ABB RAPID module: bbff74c6.mod

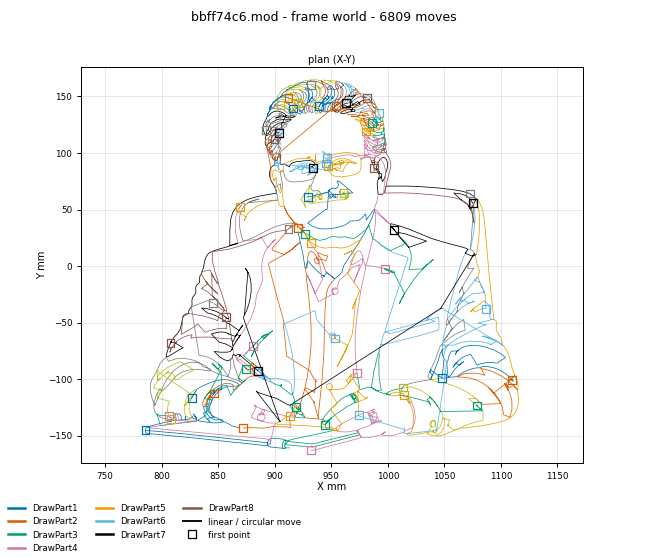
[picture p0: tool path of bbff74c6.mod in frame world, 6809 of 6811 moves have a stored position in this frame; points joined in program order, loops and branches not executed]
MODULE ImageDraw
  ! Generated 2026-10-07 06:23 for ABB IRB 1600-10/1.45: 764 strokes
  ! Page 500 x 350 mm. Work object wPaper: Z points up, so pen-up is +Z and the tool uses orientation [0,1,0,0].
  PERS tooldata tPen:=[TRUE,[[0,0,120],[1,0,0,0]],[0.3,[0,0,60],[1,0,0,0],0,0,0]];
  PERS wobjdata wPaper:=[FALSE,TRUE,"",[[700,-175,0],[1,0,0,0]],[[0,0,0],[1,0,0,0]]];
  CONST robtarget pOrigin:=[[0,0,0],[0,1,0,0],[0,0,0,0],[9E9,9E9,9E9,9E9,9E9,9E9]];
  CONST jointtarget jHome:=[[0,0,0,0,30,0],[9E9,9E9,9E9,9E9,9E9,9E9]];
  CONST speeddata vTravel:=[250,200,5000,1000];

  PROC DrawImage()
    SingArea\Wrist;
    ConfL\Off;
    ConfJ\Off;
    MoveAbsJ jHome\NoEOffs,vTravel,fine,tPen;
    DrawPart1;
    DrawPart2;
    DrawPart3;
    DrawPart4;
    DrawPart5;
    DrawPart6;
    DrawPart7;
    DrawPart8;
    DrawPart9;
    DrawPart10;
    DrawPart11;
    DrawPart12;
    DrawPart13;
    DrawPart14;
    DrawPart15;
    DrawPart16;
    DrawPart17;
    DrawPart18;
    DrawPart19;
    DrawPart20;
    DrawPart21;
    DrawPart22;
    DrawPart23;
    DrawPart24;
    DrawPart25;
    DrawPart26;
    DrawPart27;
    DrawPart28;
    DrawPart29;
    DrawPart30;
    DrawPart31;
    DrawPart32;
    DrawPart33;
    DrawPart34;
    DrawPart35;
    DrawPart36;
    DrawPart37;
    DrawPart38;
    DrawPart39;
    DrawPart40;
    DrawPart41;
    DrawPart42;
    DrawPart43;
    DrawPart44;
    DrawPart45;
    DrawPart46;
    DrawPart47;
    DrawPart48;
    DrawPart49;
    DrawPart50;
    DrawPart51;
    DrawPart52;
    DrawPart53;
    DrawPart54;
    DrawPart55;
    DrawPart56;
    DrawPart57;
    MoveAbsJ jHome\NoEOffs,vTravel,fine,tPen;
  ENDPROC

  PROC DrawPart1()
    MoveL Offs(pOrigin,85.74,29.86,6.00),vTravel,z5,tPen\WObj:=wPaper;
    MoveL Offs(pOrigin,85.74,29.86,0.00),v60,z0,tPen\WObj:=wPaper;
    MoveL Offs(pOrigin,85.74,28.38,0.00),v40,z0,tPen\WObj:=wPaper;
    MoveL Offs(pOrigin,86.16,27.45,0.00),v40,z0,tPen\WObj:=wPaper;
    MoveL Offs(pOrigin,89.14,26.89,0.00),v40,z0,tPen\WObj:=wPaper;
    MoveL Offs(pOrigin,128.88,23.06,0.00),v40,z0,tPen\WObj:=wPaper;
    MoveL Offs(pOrigin,192.62,16.26,0.00),v40,z0,tPen\WObj:=wPaper;
    MoveL Offs(pOrigin,193.90,16.48,0.00),v40,z0,tPen\WObj:=wPaper;
    MoveL Offs(pOrigin,193.90,16.48,0.00),v40,z0,tPen\WObj:=wPaper;
    MoveL Offs(pOrigin,193.90,19.02,0.00),v40,fine,tPen\WObj:=wPaper;
    MoveL Offs(pOrigin,193.90,19.02,6.00),v60,z5,tPen\WObj:=wPaper;
    MoveL Offs(pOrigin,193.90,16.48,6.00),vTravel,z5,tPen\WObj:=wPaper;
    MoveL Offs(pOrigin,193.90,16.48,0.00),v60,z0,tPen\WObj:=wPaper;
    MoveL Offs(pOrigin,195.18,15.27,0.00),v40,z0,tPen\WObj:=wPaper;
    MoveL Offs(pOrigin,206.86,14.00,0.00),v40,z0,tPen\WObj:=wPaper;
    MoveL Offs(pOrigin,207.07,15.62,0.00),v40,z0,tPen\WObj:=wPaper;
    MoveL Offs(pOrigin,206.65,16.90,0.00),v40,z0,tPen\WObj:=wPaper;
    MoveL Offs(pOrigin,207.43,19.66,0.00),v40,z0,tPen\WObj:=wPaper;
    MoveL Offs(pOrigin,208.77,21.36,0.00),v40,z0,tPen\WObj:=wPaper;
    MoveL Offs(pOrigin,208.77,21.36,0.00),v40,z0,tPen\WObj:=wPaper;
    MoveL Offs(pOrigin,207.93,22.00,0.00),v40,z0,tPen\WObj:=wPaper;
    MoveL Offs(pOrigin,199.21,22.85,0.00),v40,z0,tPen\WObj:=wPaper;
    MoveL Offs(pOrigin,196.88,22.85,0.00),v40,z0,tPen\WObj:=wPaper;
    MoveL Offs(pOrigin,194.54,21.58,0.00),v40,z0,tPen\WObj:=wPaper;
    MoveL Offs(pOrigin,194.54,21.58,0.00),v40,z0,tPen\WObj:=wPaper;
    MoveL Offs(pOrigin,193.83,19.24,0.00),v40,z0,tPen\WObj:=wPaper;
    MoveL Offs(pOrigin,192.20,19.02,0.00),v40,z0,tPen\WObj:=wPaper;
    MoveL Offs(pOrigin,118.46,26.89,0.00),v40,z0,tPen\WObj:=wPaper;
    MoveL Offs(pOrigin,85.74,29.86,0.00),v40,z0,tPen\WObj:=wPaper;
    MoveL Offs(pOrigin,85.74,29.86,0.00),v40,z0,tPen\WObj:=wPaper;
    MoveL Offs(pOrigin,86.16,31.99,0.00),v40,z0,tPen\WObj:=wPaper;
    MoveL Offs(pOrigin,88.07,32.41,0.00),v40,z0,tPen\WObj:=wPaper;
    MoveL Offs(pOrigin,88.07,32.41,0.00),v40,z0,tPen\WObj:=wPaper;
    MoveL Offs(pOrigin,88.71,33.19,0.00),v40,z0,tPen\WObj:=wPaper;
    MoveL Offs(pOrigin,96.57,35.39,0.00),v40,z0,tPen\WObj:=wPaper;
    MoveL Offs(pOrigin,105.07,37.30,0.00),v40,z0,tPen\WObj:=wPaper;
    MoveL Offs(pOrigin,107.62,37.51,0.00),v40,z0,tPen\WObj:=wPaper;
    MoveL Offs(pOrigin,108.90,38.01,0.00),v40,z0,tPen\WObj:=wPaper;
    MoveL Offs(pOrigin,109.32,38.79,0.00),v40,z0,tPen\WObj:=wPaper;
    MoveL Offs(pOrigin,109.32,38.79,0.00),v40,z0,tPen\WObj:=wPaper;
    MoveL Offs(pOrigin,108.90,39.64,0.00),v40,z0,tPen\WObj:=wPaper;
    MoveL Offs(pOrigin,108.26,39.64,0.00),v40,fine,tPen\WObj:=wPaper;
    MoveL Offs(pOrigin,108.26,39.64,6.00),v60,z5,tPen\WObj:=wPaper;
    MoveL Offs(pOrigin,109.32,38.79,6.00),vTravel,z5,tPen\WObj:=wPaper;
    MoveL Offs(pOrigin,109.32,38.79,0.00),v60,z0,tPen\WObj:=wPaper;
    MoveL Offs(pOrigin,112.72,38.72,0.00),v40,z0,tPen\WObj:=wPaper;
    MoveL Offs(pOrigin,113.08,39.21,0.00),v40,z0,tPen\WObj:=wPaper;
    MoveL Offs(pOrigin,112.51,40.70,0.00),v40,z0,tPen\WObj:=wPaper;
    MoveL Offs(pOrigin,112.51,40.70,0.00),v40,z0,tPen\WObj:=wPaper;
    MoveL Offs(pOrigin,112.37,44.53,0.00),v40,z0,tPen\WObj:=wPaper;
    MoveL Offs(pOrigin,112.94,44.74,0.00),v40,z0,tPen\WObj:=wPaper;
    MoveL Offs(pOrigin,114.21,44.10,0.00),v40,z0,tPen\WObj:=wPaper;
    MoveL Offs(pOrigin,114.21,44.10,0.00),v40,z0,tPen\WObj:=wPaper;
    MoveL Offs(pOrigin,115.49,44.38,0.00),v40,z0,tPen\WObj:=wPaper;
    MoveL Offs(pOrigin,116.34,43.67,0.00),v40,z0,tPen\WObj:=wPaper;
    MoveL Offs(pOrigin,117.26,42.19,0.00),v40,z0,tPen\WObj:=wPaper;
    MoveL Offs(pOrigin,117.82,39.42,0.00),v40,z0,tPen\WObj:=wPaper;
    MoveL Offs(pOrigin,118.25,39.00,0.00),v40,z0,tPen\WObj:=wPaper;
    MoveL Offs(pOrigin,121.22,39.42,0.00),v40,z0,tPen\WObj:=wPaper;
    MoveL Offs(pOrigin,121.01,42.61,0.00),v40,fine,tPen\WObj:=wPaper;
    MoveL Offs(pOrigin,121.01,42.61,6.00),v60,z5,tPen\WObj:=wPaper;
    MoveL Offs(pOrigin,121.44,39.42,6.00),vTravel,z5,tPen\WObj:=wPaper;
    MoveL Offs(pOrigin,121.44,39.42,0.00),v60,z0,tPen\WObj:=wPaper;
    MoveL Offs(pOrigin,122.93,39.42,0.00),v40,z0,tPen\WObj:=wPaper;
    MoveL Offs(pOrigin,123.56,39.85,0.00),v40,fine,tPen\WObj:=wPaper;
    MoveL Offs(pOrigin,123.56,39.85,6.00),v60,z5,tPen\WObj:=wPaper;
    MoveL Offs(pOrigin,127.18,41.76,6.00),vTravel,z5,tPen\WObj:=wPaper;
    MoveL Offs(pOrigin,127.18,41.76,0.00),v60,z0,tPen\WObj:=wPaper;
    MoveL Offs(pOrigin,126.96,42.19,0.00),v40,z0,tPen\WObj:=wPaper;
    MoveL Offs(pOrigin,127.18,41.76,0.00),v40,fine,tPen\WObj:=wPaper;
    MoveL Offs(pOrigin,127.18,41.76,6.00),v60,z5,tPen\WObj:=wPaper;
    MoveL Offs(pOrigin,127.81,40.28,6.00),vTravel,z5,tPen\WObj:=wPaper;
    MoveL Offs(pOrigin,127.81,40.28,0.00),v60,z0,tPen\WObj:=wPaper;
    MoveL Offs(pOrigin,130.79,39.64,0.00),v40,z0,tPen\WObj:=wPaper;
    MoveL Offs(pOrigin,130.79,39.64,0.00),v40,z0,tPen\WObj:=wPaper;
    MoveL Offs(pOrigin,130.65,41.12,0.00),v40,z0,tPen\WObj:=wPaper;
    MoveL Offs(pOrigin,128.02,44.31,0.00),v40,fine,tPen\WObj:=wPaper;
    MoveL Offs(pOrigin,128.02,44.31,6.00),v60,z5,tPen\WObj:=wPaper;
    MoveL Offs(pOrigin,129.73,41.97,6.00),vTravel,z5,tPen\WObj:=wPaper;
    MoveL Offs(pOrigin,129.73,41.97,0.00),v60,z0,tPen\WObj:=wPaper;
    MoveL Offs(pOrigin,129.51,42.40,0.00),v40,z0,tPen\WObj:=wPaper;
    MoveL Offs(pOrigin,129.73,41.97,0.00),v40,z0,tPen\WObj:=wPaper;
    MoveL Offs(pOrigin,130.36,41.34,0.00),v40,z0,tPen\WObj:=wPaper;
    MoveL Offs(pOrigin,130.15,41.76,0.00),v40,z0,tPen\WObj:=wPaper;
    MoveL Offs(pOrigin,130.36,41.34,0.00),v40,fine,tPen\WObj:=wPaper;
    MoveL Offs(pOrigin,130.36,41.34,6.00),v60,z5,tPen\WObj:=wPaper;
    MoveL Offs(pOrigin,130.79,39.64,6.00),vTravel,z5,tPen\WObj:=wPaper;
    MoveL Offs(pOrigin,130.79,39.64,0.00),v60,z0,tPen\WObj:=wPaper;
    MoveL Offs(pOrigin,131.64,38.65,0.00),v40,z0,tPen\WObj:=wPaper;
    MoveL Offs(pOrigin,134.19,37.94,0.00),v40,z0,tPen\WObj:=wPaper;
    MoveL Offs(pOrigin,141.20,36.88,0.00),v40,z0,tPen\WObj:=wPaper;
    MoveL Offs(pOrigin,142.69,36.95,0.00),v40,z0,tPen\WObj:=wPaper;
    MoveL Offs(pOrigin,142.55,37.94,0.00),v40,z0,tPen\WObj:=wPaper;
    MoveL Offs(pOrigin,140.99,39.07,0.00),v40,z0,tPen\WObj:=wPaper;
    MoveL Offs(pOrigin,138.86,41.55,0.00),v40,z0,tPen\WObj:=wPaper;
    MoveL Offs(pOrigin,136.95,45.16,0.00),v40,fine,tPen\WObj:=wPaper;
    MoveL Offs(pOrigin,136.95,45.16,6.00),v60,z5,tPen\WObj:=wPaper;
    MoveL Offs(pOrigin,139.71,45.80,6.00),vTravel,z5,tPen\WObj:=wPaper;
    MoveL Offs(pOrigin,139.71,45.80,0.00),v60,z0,tPen\WObj:=wPaper;
    MoveL Offs(pOrigin,139.93,47.08,0.00),v40,z0,tPen\WObj:=wPaper;
    MoveL Offs(pOrigin,139.50,48.99,0.00),v40,z0,tPen\WObj:=wPaper;
    MoveL Offs(pOrigin,139.50,51.11,0.00),v40,z0,tPen\WObj:=wPaper;
    MoveL Offs(pOrigin,139.50,51.11,0.00),v40,z0,tPen\WObj:=wPaper;
    MoveL Offs(pOrigin,140.99,51.04,0.00),v40,z0,tPen\WObj:=wPaper;
    MoveL Offs(pOrigin,140.77,49.41,0.00),v40,z0,tPen\WObj:=wPaper;
    MoveL Offs(pOrigin,141.70,46.01,0.00),v40,z0,tPen\WObj:=wPaper;
    MoveL Offs(pOrigin,142.90,45.59,0.00),v40,z0,tPen\WObj:=wPaper;
    MoveL Offs(pOrigin,142.90,45.59,0.00),v40,z0,tPen\WObj:=wPaper;
    MoveL Offs(pOrigin,144.18,43.25,0.00),v40,z0,tPen\WObj:=wPaper;
    MoveL Offs(pOrigin,145.24,42.19,0.00),v40,z0,tPen\WObj:=wPaper;
    MoveL Offs(pOrigin,146.51,41.48,0.00),v40,z0,tPen\WObj:=wPaper;
    MoveL Offs(pOrigin,149.70,40.63,0.00),v40,z0,tPen\WObj:=wPaper;
    MoveL Offs(pOrigin,150.34,39.64,0.00),v40,z0,tPen\WObj:=wPaper;
    MoveL Offs(pOrigin,150.34,39.64,0.00),v40,z0,tPen\WObj:=wPaper;
    MoveL Offs(pOrigin,153.10,39.28,0.00),v40,z0,tPen\WObj:=wPaper;
    MoveL Offs(pOrigin,153.88,38.79,0.00),v40,z0,tPen\WObj:=wPaper;
    MoveL Offs(pOrigin,154.59,37.58,0.00),v40,z0,tPen\WObj:=wPaper;
    MoveL Offs(pOrigin,157.14,36.73,0.00),v40,z0,tPen\WObj:=wPaper;
    MoveL Offs(pOrigin,162.66,33.62,0.00),v40,z0,tPen\WObj:=wPaper;
    MoveL Offs(pOrigin,168.82,32.20,0.00),v40,z0,tPen\WObj:=wPaper;
  ENDPROC

  PROC DrawPart2()
    MoveL Offs(pOrigin,172.01,31.99,0.00),v40,z0,tPen\WObj:=wPaper;
    MoveL Offs(pOrigin,181.15,32.20,0.00),v40,z0,tPen\WObj:=wPaper;
    MoveL Offs(pOrigin,188.80,31.77,0.00),v40,z0,tPen\WObj:=wPaper;
    MoveL Offs(pOrigin,194.11,32.20,0.00),v40,z0,tPen\WObj:=wPaper;
    MoveL Offs(pOrigin,199.43,33.69,0.00),v40,z0,tPen\WObj:=wPaper;
    MoveL Offs(pOrigin,199.43,33.69,0.00),v40,z0,tPen\WObj:=wPaper;
    MoveL Offs(pOrigin,200.27,33.05,0.00),v40,z0,tPen\WObj:=wPaper;
    MoveL Offs(pOrigin,210.48,32.84,0.00),v40,z0,tPen\WObj:=wPaper;
    MoveL Offs(pOrigin,213.88,32.41,0.00),v40,fine,tPen\WObj:=wPaper;
    MoveL Offs(pOrigin,213.88,32.41,6.00),v60,z5,tPen\WObj:=wPaper;
    MoveL Offs(pOrigin,213.02,42.19,6.00),vTravel,z5,tPen\WObj:=wPaper;
    MoveL Offs(pOrigin,213.02,42.19,0.00),v60,z0,tPen\WObj:=wPaper;
    MoveL Offs(pOrigin,215.22,44.74,0.00),v40,z0,tPen\WObj:=wPaper;
    MoveL Offs(pOrigin,215.79,46.44,0.00),v40,z0,tPen\WObj:=wPaper;
    MoveL Offs(pOrigin,215.79,47.50,0.00),v40,fine,tPen\WObj:=wPaper;
    MoveL Offs(pOrigin,215.79,47.50,6.00),v60,z5,tPen\WObj:=wPaper;
    MoveL Offs(pOrigin,218.12,50.69,6.00),vTravel,z5,tPen\WObj:=wPaper;
    MoveL Offs(pOrigin,218.12,50.69,0.00),v60,z0,tPen\WObj:=wPaper;
    MoveL Offs(pOrigin,216.00,53.03,0.00),v40,fine,tPen\WObj:=wPaper;
    MoveL Offs(pOrigin,216.00,53.03,6.00),v60,z5,tPen\WObj:=wPaper;
    MoveL Offs(pOrigin,217.06,53.66,6.00),vTravel,z5,tPen\WObj:=wPaper;
    MoveL Offs(pOrigin,217.06,53.66,0.00),v60,z0,tPen\WObj:=wPaper;
    MoveL Offs(pOrigin,220.25,50.55,0.00),v40,z0,tPen\WObj:=wPaper;
    MoveL Offs(pOrigin,221.31,50.26,0.00),v40,z0,tPen\WObj:=wPaper;
    MoveL Offs(pOrigin,221.31,50.26,0.00),v40,z0,tPen\WObj:=wPaper;
    MoveL Offs(pOrigin,222.45,52.39,0.00),v40,z0,tPen\WObj:=wPaper;
    MoveL Offs(pOrigin,226.62,66.41,0.00),v40,z0,tPen\WObj:=wPaper;
    MoveL Offs(pOrigin,228.54,75.55,0.00),v40,z0,tPen\WObj:=wPaper;
    MoveL Offs(pOrigin,229.60,82.56,0.00),v40,z0,tPen\WObj:=wPaper;
    MoveL Offs(pOrigin,230.02,83.62,0.00),v40,z0,tPen\WObj:=wPaper;
    MoveL Offs(pOrigin,231.30,94.68,0.00),v40,z0,tPen\WObj:=wPaper;
    MoveL Offs(pOrigin,232.15,105.94,0.00),v40,z0,tPen\WObj:=wPaper;
    MoveL Offs(pOrigin,232.15,121.45,0.00),v40,z0,tPen\WObj:=wPaper;
    MoveL Offs(pOrigin,231.73,129.52,0.00),v40,z0,tPen\WObj:=wPaper;
    MoveL Offs(pOrigin,230.24,146.31,0.00),v40,z0,tPen\WObj:=wPaper;
    MoveL Offs(pOrigin,227.90,165.44,0.00),v40,z0,tPen\WObj:=wPaper;
    MoveL Offs(pOrigin,228.11,167.99,0.00),v40,z0,tPen\WObj:=wPaper;
    MoveL Offs(pOrigin,227.48,170.32,0.00),v40,z0,tPen\WObj:=wPaper;
    MoveL Offs(pOrigin,227.48,172.88,0.00),v40,z0,tPen\WObj:=wPaper;
    MoveL Offs(pOrigin,227.48,172.88,0.00),v40,z0,tPen\WObj:=wPaper;
    MoveL Offs(pOrigin,228.54,173.73,0.00),v40,z0,tPen\WObj:=wPaper;
    MoveL Offs(pOrigin,228.96,179.04,0.00),v40,z0,tPen\WObj:=wPaper;
    MoveL Offs(pOrigin,228.96,179.04,0.00),v40,z0,tPen\WObj:=wPaper;
    MoveL Offs(pOrigin,229.39,184.14,0.00),v40,z0,tPen\WObj:=wPaper;
    MoveL Offs(pOrigin,230.24,186.69,0.00),v40,z0,tPen\WObj:=wPaper;
    MoveL Offs(pOrigin,231.51,187.82,0.00),v40,z0,tPen\WObj:=wPaper;
    MoveL Offs(pOrigin,232.57,187.96,0.00),v40,z0,tPen\WObj:=wPaper;
    MoveL Offs(pOrigin,234.49,186.97,0.00),v40,z0,tPen\WObj:=wPaper;
    MoveL Offs(pOrigin,237.46,182.86,0.00),v40,z0,tPen\WObj:=wPaper;
    MoveL Offs(pOrigin,237.04,182.15,0.00),v40,z0,tPen\WObj:=wPaper;
    MoveL Offs(pOrigin,238.17,180.95,0.00),v40,z0,tPen\WObj:=wPaper;
    MoveL Offs(pOrigin,238.95,178.82,0.00),v40,z0,tPen\WObj:=wPaper;
    MoveL Offs(pOrigin,238.52,176.98,0.00),v40,z0,tPen\WObj:=wPaper;
    MoveL Offs(pOrigin,237.04,177.05,0.00),v40,z0,tPen\WObj:=wPaper;
    MoveL Offs(pOrigin,235.69,178.61,0.00),v40,z0,tPen\WObj:=wPaper;
    MoveL Offs(pOrigin,235.12,180.10,0.00),v40,z0,tPen\WObj:=wPaper;
    MoveL Offs(pOrigin,235.12,181.16,0.00),v40,z0,tPen\WObj:=wPaper;
    MoveL Offs(pOrigin,235.76,182.08,0.00),v40,z0,tPen\WObj:=wPaper;
    MoveL Offs(pOrigin,237.04,182.15,0.00),v40,fine,tPen\WObj:=wPaper;
    MoveL Offs(pOrigin,237.04,182.15,6.00),v60,z5,tPen\WObj:=wPaper;
    MoveL Offs(pOrigin,237.89,181.16,6.00),vTravel,z5,tPen\WObj:=wPaper;
    MoveL Offs(pOrigin,237.89,181.16,0.00),v60,z0,tPen\WObj:=wPaper;
    MoveL Offs(pOrigin,237.04,182.01,0.00),v40,z0,tPen\WObj:=wPaper;
    MoveL Offs(pOrigin,237.89,181.16,0.00),v40,z0,tPen\WObj:=wPaper;
    MoveL Offs(pOrigin,238.31,180.31,0.00),v40,z0,tPen\WObj:=wPaper;
    MoveL Offs(pOrigin,238.10,180.74,0.00),v40,z0,tPen\WObj:=wPaper;
    MoveL Offs(pOrigin,238.31,180.31,0.00),v40,fine,tPen\WObj:=wPaper;
    MoveL Offs(pOrigin,238.31,180.31,6.00),v60,z5,tPen\WObj:=wPaper;
    MoveL Offs(pOrigin,241.29,180.95,6.00),vTravel,z5,tPen\WObj:=wPaper;
    MoveL Offs(pOrigin,241.29,180.95,0.00),v60,z0,tPen\WObj:=wPaper;
    MoveL Offs(pOrigin,238.38,185.62,0.00),v40,z0,tPen\WObj:=wPaper;
    MoveL Offs(pOrigin,238.10,186.90,0.00),v40,z0,tPen\WObj:=wPaper;
    MoveL Offs(pOrigin,238.10,186.90,0.00),v40,z0,tPen\WObj:=wPaper;
    MoveL Offs(pOrigin,243.84,184.70,0.00),v40,z0,tPen\WObj:=wPaper;
    MoveL Offs(pOrigin,247.02,183.93,0.00),v40,fine,tPen\WObj:=wPaper;
    MoveL Offs(pOrigin,247.02,183.93,6.00),v60,z5,tPen\WObj:=wPaper;
    MoveL Offs(pOrigin,245.11,179.68,6.00),vTravel,z5,tPen\WObj:=wPaper;
    MoveL Offs(pOrigin,245.11,179.68,0.00),v60,z0,tPen\WObj:=wPaper;
    MoveL Offs(pOrigin,242.35,180.88,0.00),v40,z0,tPen\WObj:=wPaper;
    MoveL Offs(pOrigin,241.29,180.95,0.00),v40,z0,tPen\WObj:=wPaper;
    MoveL Offs(pOrigin,241.29,180.95,0.00),v40,z0,tPen\WObj:=wPaper;
    MoveL Offs(pOrigin,244.83,170.96,0.00),v40,z0,tPen\WObj:=wPaper;
    MoveL Offs(pOrigin,246.81,168.62,0.00),v40,z0,tPen\WObj:=wPaper;
    MoveL Offs(pOrigin,249.36,166.71,0.00),v40,z0,tPen\WObj:=wPaper;
    MoveL Offs(pOrigin,249.79,166.50,0.00),v40,z0,tPen\WObj:=wPaper;
    MoveL Offs(pOrigin,252.98,163.74,0.00),v40,z0,tPen\WObj:=wPaper;
    MoveL Offs(pOrigin,252.98,163.74,0.00),v40,z0,tPen\WObj:=wPaper;
    MoveL Offs(pOrigin,252.55,162.89,0.00),v40,z0,tPen\WObj:=wPaper;
    MoveL Offs(pOrigin,248.94,158.85,0.00),v40,z0,tPen\WObj:=wPaper;
    MoveL Offs(pOrigin,247.17,155.66,0.00),v40,z0,tPen\WObj:=wPaper;
    MoveL Offs(pOrigin,245.96,151.41,0.00),v40,z0,tPen\WObj:=wPaper;
    MoveL Offs(pOrigin,245.32,147.16,0.00),v40,z0,tPen\WObj:=wPaper;
    MoveL Offs(pOrigin,244.48,135.69,0.00),v40,z0,tPen\WObj:=wPaper;
    MoveL Offs(pOrigin,243.41,97.01,0.00),v40,z0,tPen\WObj:=wPaper;
    MoveL Offs(pOrigin,241.93,75.34,0.00),v40,z0,tPen\WObj:=wPaper;
    MoveL Offs(pOrigin,238.95,46.86,0.00),v40,z0,tPen\WObj:=wPaper;
    MoveL Offs(pOrigin,238.74,40.28,0.00),v40,z0,tPen\WObj:=wPaper;
    MoveL Offs(pOrigin,238.52,39.99,0.00),v40,z0,tPen\WObj:=wPaper;
    MoveL Offs(pOrigin,235.55,40.06,0.00),v40,z0,tPen\WObj:=wPaper;
    MoveL Offs(pOrigin,226.41,40.91,0.00),v40,z0,tPen\WObj:=wPaper;
    MoveL Offs(pOrigin,226.41,40.91,0.00),v40,z0,tPen\WObj:=wPaper;
    MoveL Offs(pOrigin,226.41,41.76,0.00),v40,z0,tPen\WObj:=wPaper;
    MoveL Offs(pOrigin,225.99,42.40,0.00),v40,z0,tPen\WObj:=wPaper;
    MoveL Offs(pOrigin,225.99,42.40,0.00),v40,z0,tPen\WObj:=wPaper;
    MoveL Offs(pOrigin,225.70,43.67,0.00),v40,z0,tPen\WObj:=wPaper;
    MoveL Offs(pOrigin,225.14,44.45,0.00),v40,z0,tPen\WObj:=wPaper;
    MoveL Offs(pOrigin,224.71,44.53,0.00),v40,z0,tPen\WObj:=wPaper;
    MoveL Offs(pOrigin,224.71,44.53,0.00),v40,z0,tPen\WObj:=wPaper;
    MoveL Offs(pOrigin,224.29,45.59,0.00),v40,z0,tPen\WObj:=wPaper;
    MoveL Offs(pOrigin,221.60,49.20,0.00),v40,z0,tPen\WObj:=wPaper;
    MoveL Offs(pOrigin,221.31,50.26,0.00),v40,fine,tPen\WObj:=wPaper;
    MoveL Offs(pOrigin,221.31,50.26,6.00),v60,z5,tPen\WObj:=wPaper;
    MoveL Offs(pOrigin,220.04,48.78,6.00),vTravel,z5,tPen\WObj:=wPaper;
    MoveL Offs(pOrigin,220.04,48.78,0.00),v60,z0,tPen\WObj:=wPaper;
    MoveL Offs(pOrigin,219.82,49.20,0.00),v40,z0,tPen\WObj:=wPaper;
    MoveL Offs(pOrigin,220.04,48.78,0.00),v40,z0,tPen\WObj:=wPaper;
    MoveL Offs(pOrigin,220.68,48.14,0.00),v40,z0,tPen\WObj:=wPaper;
    MoveL Offs(pOrigin,220.46,48.56,0.00),v40,z0,tPen\WObj:=wPaper;
    MoveL Offs(pOrigin,220.68,48.14,0.00),v40,z0,tPen\WObj:=wPaper;
    MoveL Offs(pOrigin,221.31,47.71,0.00),v40,z0,tPen\WObj:=wPaper;
  ENDPROC

  PROC DrawPart3()
    MoveL Offs(pOrigin,218.55,50.47,0.00),v40,fine,tPen\WObj:=wPaper;
    MoveL Offs(pOrigin,218.55,50.47,6.00),v60,z5,tPen\WObj:=wPaper;
    MoveL Offs(pOrigin,219.40,49.41,6.00),vTravel,z5,tPen\WObj:=wPaper;
    MoveL Offs(pOrigin,219.40,49.41,0.00),v60,z0,tPen\WObj:=wPaper;
    MoveL Offs(pOrigin,219.19,49.84,0.00),v40,z0,tPen\WObj:=wPaper;
    MoveL Offs(pOrigin,219.40,49.41,0.00),v40,fine,tPen\WObj:=wPaper;
    MoveL Offs(pOrigin,219.40,49.41,6.00),v60,z5,tPen\WObj:=wPaper;
    MoveL Offs(pOrigin,222.16,48.35,6.00),vTravel,z5,tPen\WObj:=wPaper;
    MoveL Offs(pOrigin,222.16,48.35,0.00),v60,z0,tPen\WObj:=wPaper;
    MoveL Offs(pOrigin,221.74,48.78,0.00),v40,z0,tPen\WObj:=wPaper;
    MoveL Offs(pOrigin,222.16,48.35,0.00),v40,fine,tPen\WObj:=wPaper;
    MoveL Offs(pOrigin,222.16,48.35,6.00),v60,z5,tPen\WObj:=wPaper;
    MoveL Offs(pOrigin,219.19,44.95,6.00),vTravel,z5,tPen\WObj:=wPaper;
    MoveL Offs(pOrigin,219.19,44.95,0.00),v60,z0,tPen\WObj:=wPaper;
    MoveL Offs(pOrigin,218.12,41.55,0.00),v40,z0,tPen\WObj:=wPaper;
    MoveL Offs(pOrigin,218.12,41.55,0.00),v40,z0,tPen\WObj:=wPaper;
    MoveL Offs(pOrigin,223.23,40.91,0.00),v40,z0,tPen\WObj:=wPaper;
    MoveL Offs(pOrigin,226.41,40.91,0.00),v40,fine,tPen\WObj:=wPaper;
    MoveL Offs(pOrigin,226.41,40.91,6.00),v60,z5,tPen\WObj:=wPaper;
    MoveL Offs(pOrigin,225.99,42.40,6.00),vTravel,z5,tPen\WObj:=wPaper;
    MoveL Offs(pOrigin,225.99,42.40,0.00),v60,z0,tPen\WObj:=wPaper;
    MoveL Offs(pOrigin,224.71,42.54,0.00),v40,z0,tPen\WObj:=wPaper;
    MoveL Offs(pOrigin,223.65,43.46,0.00),v40,fine,tPen\WObj:=wPaper;
    MoveL Offs(pOrigin,223.65,43.46,6.00),v60,z5,tPen\WObj:=wPaper;
    MoveL Offs(pOrigin,224.71,44.53,6.00),vTravel,z5,tPen\WObj:=wPaper;
    MoveL Offs(pOrigin,224.71,44.53,0.00),v60,z0,tPen\WObj:=wPaper;
    MoveL Offs(pOrigin,223.23,43.53,0.00),v40,z0,tPen\WObj:=wPaper;
    MoveL Offs(pOrigin,221.10,44.60,0.00),v40,z0,tPen\WObj:=wPaper;
    MoveL Offs(pOrigin,219.40,45.02,0.00),v40,z0,tPen\WObj:=wPaper;
    MoveL Offs(pOrigin,218.76,46.01,0.00),v40,z0,tPen\WObj:=wPaper;
    MoveL Offs(pOrigin,215.86,47.71,0.00),v40,z0,tPen\WObj:=wPaper;
    MoveL Offs(pOrigin,215.50,48.78,0.00),v40,z0,tPen\WObj:=wPaper;
    MoveL Offs(pOrigin,213.73,51.11,0.00),v40,z0,tPen\WObj:=wPaper;
    MoveL Offs(pOrigin,213.45,51.96,0.00),v40,z0,tPen\WObj:=wPaper;
    MoveL Offs(pOrigin,213.45,51.96,0.00),v40,z0,tPen\WObj:=wPaper;
    MoveL Offs(pOrigin,213.66,52.32,0.00),v40,z0,tPen\WObj:=wPaper;
    MoveL Offs(pOrigin,215.36,52.74,0.00),v40,z0,tPen\WObj:=wPaper;
    MoveL Offs(pOrigin,217.06,54.09,0.00),v40,z0,tPen\WObj:=wPaper;
    MoveL Offs(pOrigin,217.49,56.85,0.00),v40,z0,tPen\WObj:=wPaper;
    MoveL Offs(pOrigin,216.00,61.31,0.00),v40,fine,tPen\WObj:=wPaper;
    MoveL Offs(pOrigin,216.00,61.31,6.00),v60,z5,tPen\WObj:=wPaper;
    MoveL Offs(pOrigin,216.00,62.80,6.00),vTravel,z5,tPen\WObj:=wPaper;
    MoveL Offs(pOrigin,216.00,62.80,0.00),v60,z0,tPen\WObj:=wPaper;
    MoveL Offs(pOrigin,215.79,61.38,0.00),v40,z0,tPen\WObj:=wPaper;
    MoveL Offs(pOrigin,214.30,61.60,0.00),v40,z0,tPen\WObj:=wPaper;
    MoveL Offs(pOrigin,205.59,68.32,0.00),v40,z0,tPen\WObj:=wPaper;
    MoveL Offs(pOrigin,205.16,68.96,0.00),v40,z0,tPen\WObj:=wPaper;
    MoveL Offs(pOrigin,205.16,68.96,0.00),v40,z0,tPen\WObj:=wPaper;
    MoveL Offs(pOrigin,206.01,70.24,0.00),v40,z0,tPen\WObj:=wPaper;
    MoveL Offs(pOrigin,205.59,69.81,0.00),v40,z0,tPen\WObj:=wPaper;
    MoveL Offs(pOrigin,206.01,70.24,0.00),v40,z0,tPen\WObj:=wPaper;
    MoveL Offs(pOrigin,205.59,69.81,0.00),v40,z0,tPen\WObj:=wPaper;
    MoveL Offs(pOrigin,205.16,68.96,0.00),v40,z0,tPen\WObj:=wPaper;
    MoveL Offs(pOrigin,200.49,70.59,0.00),v40,z0,tPen\WObj:=wPaper;
    MoveL Offs(pOrigin,196.66,72.79,0.00),v40,fine,tPen\WObj:=wPaper;
    MoveL Offs(pOrigin,196.66,72.79,6.00),v60,z5,tPen\WObj:=wPaper;
    MoveL Offs(pOrigin,195.60,75.55,6.00),vTravel,z5,tPen\WObj:=wPaper;
    MoveL Offs(pOrigin,195.60,75.55,0.00),v60,z0,tPen\WObj:=wPaper;
    MoveL Offs(pOrigin,194.11,76.19,0.00),v40,z0,tPen\WObj:=wPaper;
    MoveL Offs(pOrigin,190.07,79.45,0.00),v40,z0,tPen\WObj:=wPaper;
    MoveL Offs(pOrigin,189.30,81.29,0.00),v40,z0,tPen\WObj:=wPaper;
    MoveL Offs(pOrigin,188.38,81.71,0.00),v40,z0,tPen\WObj:=wPaper;
    MoveL Offs(pOrigin,188.38,81.71,0.00),v40,z0,tPen\WObj:=wPaper;
    MoveL Offs(pOrigin,188.16,82.49,0.00),v40,z0,tPen\WObj:=wPaper;
    MoveL Offs(pOrigin,182.43,87.66,0.00),v40,fine,tPen\WObj:=wPaper;
    MoveL Offs(pOrigin,182.43,87.66,6.00),v60,z5,tPen\WObj:=wPaper;
    MoveL Offs(pOrigin,180.94,88.72,6.00),vTravel,z5,tPen\WObj:=wPaper;
    MoveL Offs(pOrigin,180.94,88.72,0.00),v60,z0,tPen\WObj:=wPaper;
    MoveL Offs(pOrigin,181.86,87.95,0.00),v40,z0,tPen\WObj:=wPaper;
    MoveL Offs(pOrigin,172.86,95.31,0.00),v40,z0,tPen\WObj:=wPaper;
    MoveL Offs(pOrigin,172.72,95.74,0.00),v40,z0,tPen\WObj:=wPaper;
    MoveL Offs(pOrigin,176.48,99.99,0.00),v40,z0,tPen\WObj:=wPaper;
    MoveL Offs(pOrigin,190.93,114.44,0.00),v40,fine,tPen\WObj:=wPaper;
    MoveL Offs(pOrigin,190.93,114.44,6.00),v60,z5,tPen\WObj:=wPaper;
    MoveL Offs(pOrigin,193.69,114.22,6.00),vTravel,z5,tPen\WObj:=wPaper;
    MoveL Offs(pOrigin,193.69,114.22,0.00),v60,z0,tPen\WObj:=wPaper;
    MoveL Offs(pOrigin,194.11,114.65,0.00),v40,z0,tPen\WObj:=wPaper;
    MoveL Offs(pOrigin,193.69,114.22,0.00),v40,fine,tPen\WObj:=wPaper;
    MoveL Offs(pOrigin,193.69,114.22,6.00),v60,z5,tPen\WObj:=wPaper;
    MoveL Offs(pOrigin,190.50,111.25,6.00),vTravel,z5,tPen\WObj:=wPaper;
    MoveL Offs(pOrigin,190.50,111.25,0.00),v60,z0,tPen\WObj:=wPaper;
    MoveL Offs(pOrigin,192.84,113.59,0.00),v40,z0,tPen\WObj:=wPaper;
    MoveL Offs(pOrigin,190.50,111.25,0.00),v40,fine,tPen\WObj:=wPaper;
    MoveL Offs(pOrigin,190.50,111.25,6.00),v60,z5,tPen\WObj:=wPaper;
    MoveL Offs(pOrigin,188.59,112.31,6.00),vTravel,z5,tPen\WObj:=wPaper;
    MoveL Offs(pOrigin,188.59,112.31,0.00),v60,z0,tPen\WObj:=wPaper;
    MoveL Offs(pOrigin,189.65,113.38,0.00),v40,z0,tPen\WObj:=wPaper;
    MoveL Offs(pOrigin,188.59,112.31,0.00),v40,fine,tPen\WObj:=wPaper;
    MoveL Offs(pOrigin,188.59,112.31,6.00),v60,z5,tPen\WObj:=wPaper;
    MoveL Offs(pOrigin,197.51,117.41,6.00),vTravel,z5,tPen\WObj:=wPaper;
    MoveL Offs(pOrigin,197.51,117.41,0.00),v60,z0,tPen\WObj:=wPaper;
    MoveL Offs(pOrigin,197.94,117.62,0.00),v40,z0,tPen\WObj:=wPaper;
    MoveL Offs(pOrigin,197.51,117.41,0.00),v40,z0,tPen\WObj:=wPaper;
    MoveL Offs(pOrigin,197.94,117.62,0.00),v40,z0,tPen\WObj:=wPaper;
    MoveL Offs(pOrigin,193.05,113.59,0.00),v40,z0,tPen\WObj:=wPaper;
    MoveL Offs(pOrigin,187.31,107.64,0.00),v40,z0,tPen\WObj:=wPaper;
    MoveL Offs(pOrigin,182.35,100.62,0.00),v40,z0,tPen\WObj:=wPaper;
    MoveL Offs(pOrigin,179.24,94.68,0.00),v40,z0,tPen\WObj:=wPaper;
    MoveL Offs(pOrigin,179.45,95.53,0.00),v40,z0,tPen\WObj:=wPaper;
    MoveL Offs(pOrigin,179.66,95.95,0.00),v40,z0,tPen\WObj:=wPaper;
    MoveL Offs(pOrigin,179.45,95.53,0.00),v40,fine,tPen\WObj:=wPaper;
    MoveL Offs(pOrigin,179.45,95.53,6.00),v60,z5,tPen\WObj:=wPaper;
    MoveL Offs(pOrigin,180.51,97.65,6.00),vTravel,z5,tPen\WObj:=wPaper;
    MoveL Offs(pOrigin,180.51,97.65,0.00),v60,z0,tPen\WObj:=wPaper;
    MoveL Offs(pOrigin,180.73,98.07,0.00),v40,z0,tPen\WObj:=wPaper;
    MoveL Offs(pOrigin,180.51,97.65,0.00),v40,fine,tPen\WObj:=wPaper;
    MoveL Offs(pOrigin,180.51,97.65,6.00),v60,z5,tPen\WObj:=wPaper;
    MoveL Offs(pOrigin,181.36,99.14,6.00),vTravel,z5,tPen\WObj:=wPaper;
    MoveL Offs(pOrigin,181.36,99.14,0.00),v60,z0,tPen\WObj:=wPaper;
    MoveL Offs(pOrigin,181.57,99.56,0.00),v40,z0,tPen\WObj:=wPaper;
    MoveL Offs(pOrigin,181.36,99.14,0.00),v40,fine,tPen\WObj:=wPaper;
    MoveL Offs(pOrigin,181.36,99.14,6.00),v60,z5,tPen\WObj:=wPaper;
    MoveL Offs(pOrigin,182.00,100.20,6.00),vTravel,z5,tPen\WObj:=wPaper;
    MoveL Offs(pOrigin,182.00,100.20,0.00),v60,z0,tPen\WObj:=wPaper;
    MoveL Offs(pOrigin,182.21,100.62,0.00),v40,z0,tPen\WObj:=wPaper;
    MoveL Offs(pOrigin,182.00,100.20,0.00),v40,fine,tPen\WObj:=wPaper;
    MoveL Offs(pOrigin,182.00,100.20,6.00),v60,z5,tPen\WObj:=wPaper;
    MoveL Offs(pOrigin,180.94,104.66,6.00),vTravel,z5,tPen\WObj:=wPaper;
    MoveL Offs(pOrigin,180.94,104.66,0.00),v60,z0,tPen\WObj:=wPaper;
    MoveL Offs(pOrigin,185.82,109.55,0.00),v40,z0,tPen\WObj:=wPaper;
  ENDPROC

  PROC DrawPart4()
    MoveL Offs(pOrigin,180.94,104.66,0.00),v40,fine,tPen\WObj:=wPaper;
    MoveL Offs(pOrigin,180.94,104.66,6.00),v60,z5,tPen\WObj:=wPaper;
    MoveL Offs(pOrigin,175.62,99.14,6.00),vTravel,z5,tPen\WObj:=wPaper;
    MoveL Offs(pOrigin,175.62,99.14,0.00),v60,z0,tPen\WObj:=wPaper;
    MoveL Offs(pOrigin,176.05,99.56,0.00),v40,z0,tPen\WObj:=wPaper;
    MoveL Offs(pOrigin,175.62,99.14,0.00),v40,fine,tPen\WObj:=wPaper;
    MoveL Offs(pOrigin,175.62,99.14,6.00),v60,z5,tPen\WObj:=wPaper;
    MoveL Offs(pOrigin,174.14,97.65,6.00),vTravel,z5,tPen\WObj:=wPaper;
    MoveL Offs(pOrigin,174.14,97.65,0.00),v60,z0,tPen\WObj:=wPaper;
    MoveL Offs(pOrigin,174.99,98.50,0.00),v40,z0,tPen\WObj:=wPaper;
    MoveL Offs(pOrigin,174.14,97.65,0.00),v40,fine,tPen\WObj:=wPaper;
    MoveL Offs(pOrigin,174.14,97.65,6.00),v60,z5,tPen\WObj:=wPaper;
    MoveL Offs(pOrigin,172.65,95.95,6.00),vTravel,z5,tPen\WObj:=wPaper;
    MoveL Offs(pOrigin,172.65,95.95,0.00),v60,z0,tPen\WObj:=wPaper;
    MoveL Offs(pOrigin,169.68,96.59,0.00),v40,z0,tPen\WObj:=wPaper;
    MoveL Offs(pOrigin,169.68,96.59,0.00),v40,z0,tPen\WObj:=wPaper;
    MoveL Offs(pOrigin,167.98,94.46,0.00),v40,z0,tPen\WObj:=wPaper;
    MoveL Offs(pOrigin,166.49,93.40,0.00),v40,z0,tPen\WObj:=wPaper;
    MoveL Offs(pOrigin,166.49,93.40,0.00),v40,z0,tPen\WObj:=wPaper;
    MoveL Offs(pOrigin,167.98,91.06,0.00),v40,z0,tPen\WObj:=wPaper;
    MoveL Offs(pOrigin,180.73,79.45,0.00),v40,z0,tPen\WObj:=wPaper;
    MoveL Offs(pOrigin,181.57,77.96,0.00),v40,z0,tPen\WObj:=wPaper;
    MoveL Offs(pOrigin,184.98,77.04,0.00),v40,z0,tPen\WObj:=wPaper;
    MoveL Offs(pOrigin,186.18,77.04,0.00),v40,z0,tPen\WObj:=wPaper;
    MoveL Offs(pOrigin,186.18,78.10,0.00),v40,z0,tPen\WObj:=wPaper;
    MoveL Offs(pOrigin,176.90,86.39,0.00),v40,fine,tPen\WObj:=wPaper;
    MoveL Offs(pOrigin,176.90,86.39,6.00),v60,z5,tPen\WObj:=wPaper;
    MoveL Offs(pOrigin,175.84,87.03,6.00),vTravel,z5,tPen\WObj:=wPaper;
    MoveL Offs(pOrigin,175.84,87.03,0.00),v60,z0,tPen\WObj:=wPaper;
    MoveL Offs(pOrigin,176.33,86.67,0.00),v40,z0,tPen\WObj:=wPaper;
    MoveL Offs(pOrigin,169.25,92.76,0.00),v40,fine,tPen\WObj:=wPaper;
    MoveL Offs(pOrigin,169.25,92.76,6.00),v60,z5,tPen\WObj:=wPaper;
    MoveL Offs(pOrigin,167.55,91.49,6.00),vTravel,z5,tPen\WObj:=wPaper;
    MoveL Offs(pOrigin,167.55,91.49,0.00),v60,z0,tPen\WObj:=wPaper;
    MoveL Offs(pOrigin,167.34,91.91,0.00),v40,z0,tPen\WObj:=wPaper;
    MoveL Offs(pOrigin,167.55,91.49,0.00),v40,z0,tPen\WObj:=wPaper;
    MoveL Offs(pOrigin,167.12,92.12,0.00),v40,z0,tPen\WObj:=wPaper;
    MoveL Offs(pOrigin,166.70,92.55,0.00),v40,z0,tPen\WObj:=wPaper;
    MoveL Offs(pOrigin,167.12,92.12,0.00),v40,fine,tPen\WObj:=wPaper;
    MoveL Offs(pOrigin,167.12,92.12,6.00),v60,z5,tPen\WObj:=wPaper;
    MoveL Offs(pOrigin,166.49,93.40,6.00),vTravel,z5,tPen\WObj:=wPaper;
    MoveL Offs(pOrigin,166.49,93.40,0.00),v60,z0,tPen\WObj:=wPaper;
    MoveL Offs(pOrigin,165.78,94.04,0.00),v40,z0,tPen\WObj:=wPaper;
    MoveL Offs(pOrigin,165.64,95.53,0.00),v40,z0,tPen\WObj:=wPaper;
    MoveL Offs(pOrigin,165.64,95.53,0.00),v40,z0,tPen\WObj:=wPaper;
    MoveL Offs(pOrigin,163.65,97.22,0.00),v40,z0,tPen\WObj:=wPaper;
    MoveL Offs(pOrigin,163.30,101.26,0.00),v40,z0,tPen\WObj:=wPaper;
    MoveL Offs(pOrigin,162.88,101.90,0.00),v40,z0,tPen\WObj:=wPaper;
    MoveL Offs(pOrigin,162.88,101.90,0.00),v40,z0,tPen\WObj:=wPaper;
    MoveL Offs(pOrigin,162.88,103.18,0.00),v40,z0,tPen\WObj:=wPaper;
    MoveL Offs(pOrigin,162.88,103.18,0.00),v40,z0,tPen\WObj:=wPaper;
    MoveL Offs(pOrigin,166.20,108.91,0.00),v40,z0,tPen\WObj:=wPaper;
    MoveL Offs(pOrigin,175.27,122.09,0.00),v40,z0,tPen\WObj:=wPaper;
    MoveL Offs(pOrigin,179.52,130.16,0.00),v40,z0,tPen\WObj:=wPaper;
    MoveL Offs(pOrigin,182.64,139.51,0.00),v40,z0,tPen\WObj:=wPaper;
    MoveL Offs(pOrigin,183.91,149.07,0.00),v40,fine,tPen\WObj:=wPaper;
    MoveL Offs(pOrigin,183.91,149.07,6.00),v60,z5,tPen\WObj:=wPaper;
    MoveL Offs(pOrigin,189.44,162.25,6.00),vTravel,z5,tPen\WObj:=wPaper;
    MoveL Offs(pOrigin,189.44,162.25,0.00),v60,z0,tPen\WObj:=wPaper;
    MoveL Offs(pOrigin,188.59,171.18,0.00),v40,z0,tPen\WObj:=wPaper;
    MoveL Offs(pOrigin,188.59,177.12,0.00),v40,z0,tPen\WObj:=wPaper;
    MoveL Offs(pOrigin,189.65,182.86,0.00),v40,z0,tPen\WObj:=wPaper;
    MoveL Offs(pOrigin,191.28,187.32,0.00),v40,z0,tPen\WObj:=wPaper;
    MoveL Offs(pOrigin,193.26,190.51,0.00),v40,z0,tPen\WObj:=wPaper;
    MoveL Offs(pOrigin,196.66,194.76,0.00),v40,z0,tPen\WObj:=wPaper;
    MoveL Offs(pOrigin,200.91,198.59,0.00),v40,z0,tPen\WObj:=wPaper;
    MoveL Offs(pOrigin,200.49,198.38,0.00),v40,z0,tPen\WObj:=wPaper;
    MoveL Offs(pOrigin,200.91,198.59,0.00),v40,z0,tPen\WObj:=wPaper;
    MoveL Offs(pOrigin,200.49,198.38,0.00),v40,fine,tPen\WObj:=wPaper;
    MoveL Offs(pOrigin,200.49,198.38,6.00),v60,z5,tPen\WObj:=wPaper;
    MoveL Offs(pOrigin,199.21,197.31,6.00),vTravel,z5,tPen\WObj:=wPaper;
    MoveL Offs(pOrigin,199.21,197.31,0.00),v60,z0,tPen\WObj:=wPaper;
    MoveL Offs(pOrigin,199.64,197.74,0.00),v40,z0,tPen\WObj:=wPaper;
    MoveL Offs(pOrigin,199.21,197.31,0.00),v40,fine,tPen\WObj:=wPaper;
    MoveL Offs(pOrigin,199.21,197.31,6.00),v60,z5,tPen\WObj:=wPaper;
    MoveL Offs(pOrigin,198.15,196.25,6.00),vTravel,z5,tPen\WObj:=wPaper;
    MoveL Offs(pOrigin,198.15,196.25,0.00),v60,z0,tPen\WObj:=wPaper;
    MoveL Offs(pOrigin,199.00,197.10,0.00),v40,z0,tPen\WObj:=wPaper;
    MoveL Offs(pOrigin,198.15,196.25,0.00),v40,fine,tPen\WObj:=wPaper;
    MoveL Offs(pOrigin,198.15,196.25,6.00),v60,z5,tPen\WObj:=wPaper;
    MoveL Offs(pOrigin,193.69,191.36,6.00),vTravel,z5,tPen\WObj:=wPaper;
    MoveL Offs(pOrigin,193.69,191.36,0.00),v60,z0,tPen\WObj:=wPaper;
    MoveL Offs(pOrigin,194.11,191.79,0.00),v40,z0,tPen\WObj:=wPaper;
    MoveL Offs(pOrigin,193.69,191.36,0.00),v40,fine,tPen\WObj:=wPaper;
    MoveL Offs(pOrigin,193.69,191.36,6.00),v60,z5,tPen\WObj:=wPaper;
    MoveL Offs(pOrigin,188.38,200.50,6.00),vTravel,z5,tPen\WObj:=wPaper;
    MoveL Offs(pOrigin,188.38,200.50,0.00),v60,z0,tPen\WObj:=wPaper;
    MoveL Offs(pOrigin,188.80,200.71,0.00),v40,z0,tPen\WObj:=wPaper;
    MoveL Offs(pOrigin,188.38,200.50,0.00),v40,fine,tPen\WObj:=wPaper;
    MoveL Offs(pOrigin,188.38,200.50,6.00),v60,z5,tPen\WObj:=wPaper;
    MoveL Offs(pOrigin,187.10,199.86,6.00),vTravel,z5,tPen\WObj:=wPaper;
    MoveL Offs(pOrigin,187.10,199.86,0.00),v60,z0,tPen\WObj:=wPaper;
    MoveL Offs(pOrigin,187.52,200.07,0.00),v40,z0,tPen\WObj:=wPaper;
    MoveL Offs(pOrigin,187.10,199.86,0.00),v40,z0,tPen\WObj:=wPaper;
    MoveL Offs(pOrigin,186.25,199.44,0.00),v40,z0,tPen\WObj:=wPaper;
    MoveL Offs(pOrigin,186.68,199.65,0.00),v40,z0,tPen\WObj:=wPaper;
    MoveL Offs(pOrigin,186.25,199.44,0.00),v40,fine,tPen\WObj:=wPaper;
    MoveL Offs(pOrigin,186.25,199.44,6.00),v60,z5,tPen\WObj:=wPaper;
    MoveL Offs(pOrigin,184.98,198.80,6.00),vTravel,z5,tPen\WObj:=wPaper;
    MoveL Offs(pOrigin,184.98,198.80,0.00),v60,z0,tPen\WObj:=wPaper;
    MoveL Offs(pOrigin,185.40,199.01,0.00),v40,z0,tPen\WObj:=wPaper;
    MoveL Offs(pOrigin,184.98,198.80,0.00),v40,fine,tPen\WObj:=wPaper;
    MoveL Offs(pOrigin,184.98,198.80,6.00),v60,z5,tPen\WObj:=wPaper;
    MoveL Offs(pOrigin,172.01,197.10,6.00),vTravel,z5,tPen\WObj:=wPaper;
    MoveL Offs(pOrigin,172.01,197.10,0.00),v60,z0,tPen\WObj:=wPaper;
    MoveL Offs(pOrigin,171.59,196.53,0.00),v40,z0,tPen\WObj:=wPaper;
    MoveL Offs(pOrigin,169.04,195.61,0.00),v40,z0,tPen\WObj:=wPaper;
    MoveL Offs(pOrigin,167.76,195.40,0.00),v40,z0,tPen\WObj:=wPaper;
    MoveL Offs(pOrigin,167.41,195.61,0.00),v40,z0,tPen\WObj:=wPaper;
    MoveL Offs(pOrigin,165.64,203.69,0.00),v40,z0,tPen\WObj:=wPaper;
    MoveL Offs(pOrigin,165.21,207.73,0.00),v40,z0,tPen\WObj:=wPaper;
    MoveL Offs(pOrigin,165.21,216.01,0.00),v40,z0,tPen\WObj:=wPaper;
    MoveL Offs(pOrigin,165.64,218.56,0.00),v40,z0,tPen\WObj:=wPaper;
    MoveL Offs(pOrigin,167.69,224.73,0.00),v40,z0,tPen\WObj:=wPaper;
    MoveL Offs(pOrigin,170.52,228.98,0.00),v40,fine,tPen\WObj:=wPaper;
    MoveL Offs(pOrigin,170.52,228.98,6.00),v60,z5,tPen\WObj:=wPaper;
    MoveL Offs(pOrigin,169.04,227.06,6.00),vTravel,z5,tPen\WObj:=wPaper;
    MoveL Offs(pOrigin,169.04,227.06,0.00),v60,z0,tPen\WObj:=wPaper;
    MoveL Offs(pOrigin,169.46,227.70,0.00),v40,z0,tPen\WObj:=wPaper;
    MoveL Offs(pOrigin,169.04,227.06,0.00),v40,fine,tPen\WObj:=wPaper;
  ENDPROC

  PROC DrawPart5()
    MoveL Offs(pOrigin,169.04,227.06,6.00),v60,z5,tPen\WObj:=wPaper;
    MoveL Offs(pOrigin,166.91,223.24,6.00),vTravel,z5,tPen\WObj:=wPaper;
    MoveL Offs(pOrigin,166.91,223.24,0.00),v60,z0,tPen\WObj:=wPaper;
    MoveL Offs(pOrigin,167.12,223.66,0.00),v40,z0,tPen\WObj:=wPaper;
    MoveL Offs(pOrigin,166.91,223.24,0.00),v40,fine,tPen\WObj:=wPaper;
    MoveL Offs(pOrigin,166.91,223.24,6.00),v60,z5,tPen\WObj:=wPaper;
    MoveL Offs(pOrigin,174.56,218.56,6.00),vTravel,z5,tPen\WObj:=wPaper;
    MoveL Offs(pOrigin,174.56,218.56,0.00),v60,z0,tPen\WObj:=wPaper;
    MoveL Offs(pOrigin,174.77,218.99,0.00),v40,z0,tPen\WObj:=wPaper;
    MoveL Offs(pOrigin,174.56,218.56,0.00),v40,fine,tPen\WObj:=wPaper;
    MoveL Offs(pOrigin,174.56,218.56,6.00),v60,z5,tPen\WObj:=wPaper;
    MoveL Offs(pOrigin,173.29,215.38,6.00),vTravel,z5,tPen\WObj:=wPaper;
    MoveL Offs(pOrigin,173.29,215.38,0.00),v60,z0,tPen\WObj:=wPaper;
    MoveL Offs(pOrigin,174.28,218.35,0.00),v40,z0,tPen\WObj:=wPaper;
    MoveL Offs(pOrigin,175.84,220.90,0.00),v40,z0,tPen\WObj:=wPaper;
    MoveL Offs(pOrigin,179.24,224.51,0.00),v40,z0,tPen\WObj:=wPaper;
    MoveL Offs(pOrigin,182.00,226.50,0.00),v40,z0,tPen\WObj:=wPaper;
    MoveL Offs(pOrigin,185.82,228.62,0.00),v40,z0,tPen\WObj:=wPaper;
    MoveL Offs(pOrigin,190.50,230.53,0.00),v40,z0,tPen\WObj:=wPaper;
    MoveL Offs(pOrigin,197.51,232.59,0.00),v40,z0,tPen\WObj:=wPaper;
    MoveL Offs(pOrigin,202.82,233.44,0.00),v40,z0,tPen\WObj:=wPaper;
    MoveL Offs(pOrigin,202.82,233.44,0.00),v40,z0,tPen\WObj:=wPaper;
    MoveL Offs(pOrigin,203.53,230.46,0.00),v40,z0,tPen\WObj:=wPaper;
    MoveL Offs(pOrigin,204.52,228.76,0.00),v40,z0,tPen\WObj:=wPaper;
    MoveL Offs(pOrigin,206.23,227.70,0.00),v40,z0,tPen\WObj:=wPaper;
    MoveL Offs(pOrigin,208.35,227.70,0.00),v40,z0,tPen\WObj:=wPaper;
    MoveL Offs(pOrigin,208.35,227.70,0.00),v40,z0,tPen\WObj:=wPaper;
    MoveL Offs(pOrigin,207.50,231.95,0.00),v40,z0,tPen\WObj:=wPaper;
    MoveL Offs(pOrigin,207.07,237.26,0.00),v40,fine,tPen\WObj:=wPaper;
    MoveL Offs(pOrigin,207.07,237.26,6.00),v60,z5,tPen\WObj:=wPaper;
    MoveL Offs(pOrigin,206.65,240.24,6.00),vTravel,z5,tPen\WObj:=wPaper;
    MoveL Offs(pOrigin,206.65,240.24,0.00),v60,z0,tPen\WObj:=wPaper;
    MoveL Offs(pOrigin,206.44,242.36,0.00),v40,fine,tPen\WObj:=wPaper;
    MoveL Offs(pOrigin,206.44,242.36,6.00),v60,z5,tPen\WObj:=wPaper;
    MoveL Offs(pOrigin,204.95,239.60,6.00),vTravel,z5,tPen\WObj:=wPaper;
    MoveL Offs(pOrigin,204.95,239.60,0.00),v60,z0,tPen\WObj:=wPaper;
    MoveL Offs(pOrigin,201.55,247.89,0.00),v40,z0,tPen\WObj:=wPaper;
    MoveL Offs(pOrigin,201.34,253.41,0.00),v40,fine,tPen\WObj:=wPaper;
    MoveL Offs(pOrigin,201.34,253.41,6.00),v60,z5,tPen\WObj:=wPaper;
    MoveL Offs(pOrigin,199.43,251.07,6.00),vTravel,z5,tPen\WObj:=wPaper;
    MoveL Offs(pOrigin,199.43,251.07,0.00),v60,z0,tPen\WObj:=wPaper;
    MoveL Offs(pOrigin,199.21,251.50,0.00),v40,z0,tPen\WObj:=wPaper;
    MoveL Offs(pOrigin,199.43,251.07,0.00),v40,z0,tPen\WObj:=wPaper;
    MoveL Offs(pOrigin,200.06,250.23,0.00),v40,z0,tPen\WObj:=wPaper;
    MoveL Offs(pOrigin,198.72,252.77,0.00),v40,z0,tPen\WObj:=wPaper;
    MoveL Offs(pOrigin,198.15,254.69,0.00),v40,z0,tPen\WObj:=wPaper;
    MoveL Offs(pOrigin,198.15,257.02,0.00),v40,z0,tPen\WObj:=wPaper;
    MoveL Offs(pOrigin,199.07,259.79,0.00),v40,z0,tPen\WObj:=wPaper;
    MoveL Offs(pOrigin,200.06,260.00,0.00),v40,z0,tPen\WObj:=wPaper;
    MoveL Offs(pOrigin,201.12,259.72,0.00),v40,z0,tPen\WObj:=wPaper;
    MoveL Offs(pOrigin,204.74,257.88,0.00),v40,z0,tPen\WObj:=wPaper;
    MoveL Offs(pOrigin,205.16,258.30,0.00),v40,z0,tPen\WObj:=wPaper;
    MoveL Offs(pOrigin,205.16,259.36,0.00),v40,z0,tPen\WObj:=wPaper;
    MoveL Offs(pOrigin,205.16,259.36,0.00),v40,z0,tPen\WObj:=wPaper;
    MoveL Offs(pOrigin,207.07,259.58,0.00),v40,z0,tPen\WObj:=wPaper;
    MoveL Offs(pOrigin,207.07,259.36,0.00),v40,z0,tPen\WObj:=wPaper;
    MoveL Offs(pOrigin,207.07,259.36,0.00),v40,z0,tPen\WObj:=wPaper;
    MoveL Offs(pOrigin,207.50,260.21,0.00),v40,z0,tPen\WObj:=wPaper;
    MoveL Offs(pOrigin,207.50,263.40,0.00),v40,z0,tPen\WObj:=wPaper;
    MoveL Offs(pOrigin,208.14,265.31,0.00),v40,z0,tPen\WObj:=wPaper;
    MoveL Offs(pOrigin,208.14,265.31,0.00),v40,z0,tPen\WObj:=wPaper;
    MoveL Offs(pOrigin,210.69,266.87,0.00),v40,z0,tPen\WObj:=wPaper;
    MoveL Offs(pOrigin,215.79,268.43,0.00),v40,z0,tPen\WObj:=wPaper;
    MoveL Offs(pOrigin,218.34,269.56,0.00),v40,z0,tPen\WObj:=wPaper;
    MoveL Offs(pOrigin,224.93,270.41,0.00),v40,z0,tPen\WObj:=wPaper;
    MoveL Offs(pOrigin,227.48,270.41,0.00),v40,z0,tPen\WObj:=wPaper;
    MoveL Offs(pOrigin,230.02,271.48,0.00),v40,z0,tPen\WObj:=wPaper;
    MoveL Offs(pOrigin,230.02,271.48,0.00),v40,z0,tPen\WObj:=wPaper;
    MoveL Offs(pOrigin,230.24,271.90,0.00),v40,z0,tPen\WObj:=wPaper;
    MoveL Offs(pOrigin,231.73,271.48,0.00),v40,z0,tPen\WObj:=wPaper;
    MoveL Offs(pOrigin,231.30,270.84,0.00),v40,z0,tPen\WObj:=wPaper;
    MoveL Offs(pOrigin,230.02,271.05,0.00),v40,z0,tPen\WObj:=wPaper;
    MoveL Offs(pOrigin,230.02,271.05,0.00),v40,z0,tPen\WObj:=wPaper;
    MoveL Offs(pOrigin,229.60,269.99,0.00),v40,z0,tPen\WObj:=wPaper;
    MoveL Offs(pOrigin,229.60,269.99,0.00),v40,z0,tPen\WObj:=wPaper;
    MoveL Offs(pOrigin,229.60,270.20,0.00),v40,z0,tPen\WObj:=wPaper;
    MoveL Offs(pOrigin,228.96,269.99,0.00),v40,z0,tPen\WObj:=wPaper;
    MoveL Offs(pOrigin,228.54,270.62,0.00),v40,fine,tPen\WObj:=wPaper;
    MoveL Offs(pOrigin,228.54,270.62,6.00),v60,z5,tPen\WObj:=wPaper;
    MoveL Offs(pOrigin,229.60,269.99,6.00),vTravel,z5,tPen\WObj:=wPaper;
    MoveL Offs(pOrigin,229.60,269.99,0.00),v60,z0,tPen\WObj:=wPaper;
    MoveL Offs(pOrigin,235.55,268.50,0.00),v40,z0,tPen\WObj:=wPaper;
    MoveL Offs(pOrigin,235.98,269.14,0.00),v40,z0,tPen\WObj:=wPaper;
    MoveL Offs(pOrigin,235.55,268.29,0.00),v40,z0,tPen\WObj:=wPaper;
    MoveL Offs(pOrigin,236.19,267.65,0.00),v40,z0,tPen\WObj:=wPaper;
    MoveL Offs(pOrigin,236.19,267.65,0.00),v40,z0,tPen\WObj:=wPaper;
    MoveL Offs(pOrigin,236.61,268.50,0.00),v40,z0,tPen\WObj:=wPaper;
    MoveL Offs(pOrigin,235.98,269.56,0.00),v40,z0,tPen\WObj:=wPaper;
    MoveL Offs(pOrigin,236.19,274.24,0.00),v40,fine,tPen\WObj:=wPaper;
    MoveL Offs(pOrigin,236.19,274.24,6.00),v60,z5,tPen\WObj:=wPaper;
    MoveL Offs(pOrigin,236.19,267.65,6.00),vTravel,z5,tPen\WObj:=wPaper;
    MoveL Offs(pOrigin,236.19,267.65,0.00),v60,z0,tPen\WObj:=wPaper;
    MoveL Offs(pOrigin,236.82,266.59,0.00),v40,z0,tPen\WObj:=wPaper;
    MoveL Offs(pOrigin,241.50,267.86,0.00),v40,z0,tPen\WObj:=wPaper;
    MoveL Offs(pOrigin,244.90,267.65,0.00),v40,z0,tPen\WObj:=wPaper;
    MoveL Offs(pOrigin,245.25,267.86,0.00),v40,z0,tPen\WObj:=wPaper;
    MoveL Offs(pOrigin,245.75,269.70,0.00),v40,z0,tPen\WObj:=wPaper;
    MoveL Offs(pOrigin,250.43,273.03,0.00),v40,z0,tPen\WObj:=wPaper;
    MoveL Offs(pOrigin,254.04,274.24,0.00),v40,z0,tPen\WObj:=wPaper;
    MoveL Offs(pOrigin,261.05,275.30,0.00),v40,z0,tPen\WObj:=wPaper;
    MoveL Offs(pOrigin,264.24,275.51,0.00),v40,z0,tPen\WObj:=wPaper;
    MoveL Offs(pOrigin,271.89,274.45,0.00),v40,z0,tPen\WObj:=wPaper;
    MoveL Offs(pOrigin,274.01,273.67,0.00),v40,z0,tPen\WObj:=wPaper;
    MoveL Offs(pOrigin,275.08,272.75,0.00),v40,z0,tPen\WObj:=wPaper;
    MoveL Offs(pOrigin,275.08,272.75,0.00),v40,z0,tPen\WObj:=wPaper;
    MoveL Offs(pOrigin,276.00,269.56,0.00),v40,z0,tPen\WObj:=wPaper;
    MoveL Offs(pOrigin,276.35,269.35,0.00),v40,z0,tPen\WObj:=wPaper;
    MoveL Offs(pOrigin,276.35,269.35,0.00),v40,z0,tPen\WObj:=wPaper;
    MoveL Offs(pOrigin,276.35,262.34,0.00),v40,z0,tPen\WObj:=wPaper;
    MoveL Offs(pOrigin,275.57,259.36,0.00),v40,z0,tPen\WObj:=wPaper;
    MoveL Offs(pOrigin,274.86,258.09,0.00),v40,z0,tPen\WObj:=wPaper;
    MoveL Offs(pOrigin,273.16,256.95,0.00),v40,z0,tPen\WObj:=wPaper;
    MoveL Offs(pOrigin,271.04,256.10,0.00),v40,z0,tPen\WObj:=wPaper;
    MoveL Offs(pOrigin,266.36,254.90,0.00),v40,z0,tPen\WObj:=wPaper;
    MoveL Offs(pOrigin,260.20,254.05,0.00),v40,z0,tPen\WObj:=wPaper;
    MoveL Offs(pOrigin,254.89,254.05,0.00),v40,z0,tPen\WObj:=wPaper;
    MoveL Offs(pOrigin,251.91,254.83,0.00),v40,z0,tPen\WObj:=wPaper;
    MoveL Offs(pOrigin,249.57,256.81,0.00),v40,z0,tPen\WObj:=wPaper;
    MoveL Offs(pOrigin,246.53,261.06,0.00),v40,z0,tPen\WObj:=wPaper;
    MoveL Offs(pOrigin,245.54,263.83,0.00),v40,z0,tPen\WObj:=wPaper;
  ENDPROC

  PROC DrawPart6()
    MoveL Offs(pOrigin,245.25,265.74,0.00),v40,z0,tPen\WObj:=wPaper;
    MoveL Offs(pOrigin,244.26,266.16,0.00),v40,z0,tPen\WObj:=wPaper;
    MoveL Offs(pOrigin,241.93,266.38,0.00),v40,z0,tPen\WObj:=wPaper;
    MoveL Offs(pOrigin,238.10,265.38,0.00),v40,z0,tPen\WObj:=wPaper;
    MoveL Offs(pOrigin,237.25,264.46,0.00),v40,z0,tPen\WObj:=wPaper;
    MoveL Offs(pOrigin,237.25,262.98,0.00),v40,z0,tPen\WObj:=wPaper;
    MoveL Offs(pOrigin,237.68,262.55,0.00),v40,z0,tPen\WObj:=wPaper;
    MoveL Offs(pOrigin,237.68,262.55,0.00),v40,z0,tPen\WObj:=wPaper;
    MoveL Offs(pOrigin,238.10,262.98,0.00),v40,z0,tPen\WObj:=wPaper;
    MoveL Offs(pOrigin,238.10,263.83,0.00),v40,fine,tPen\WObj:=wPaper;
    MoveL Offs(pOrigin,238.10,263.83,6.00),v60,z5,tPen\WObj:=wPaper;
    MoveL Offs(pOrigin,237.68,262.12,6.00),vTravel,z5,tPen\WObj:=wPaper;
    MoveL Offs(pOrigin,237.68,262.12,0.00),v60,z0,tPen\WObj:=wPaper;
    MoveL Offs(pOrigin,237.89,260.64,0.00),v40,z0,tPen\WObj:=wPaper;
    MoveL Offs(pOrigin,237.46,260.21,0.00),v40,z0,tPen\WObj:=wPaper;
    MoveL Offs(pOrigin,237.46,260.21,0.00),v40,z0,tPen\WObj:=wPaper;
    MoveL Offs(pOrigin,236.61,257.45,0.00),v40,z0,tPen\WObj:=wPaper;
    MoveL Offs(pOrigin,236.61,257.45,0.00),v40,z0,tPen\WObj:=wPaper;
    MoveL Offs(pOrigin,236.82,257.02,0.00),v40,z0,tPen\WObj:=wPaper;
    MoveL Offs(pOrigin,237.04,257.45,0.00),v40,z0,tPen\WObj:=wPaper;
    MoveL Offs(pOrigin,237.04,257.45,0.00),v40,z0,tPen\WObj:=wPaper;
    MoveL Offs(pOrigin,237.46,257.45,0.00),v40,z0,tPen\WObj:=wPaper;
    MoveL Offs(pOrigin,237.25,258.73,0.00),v40,fine,tPen\WObj:=wPaper;
    MoveL Offs(pOrigin,237.25,258.73,6.00),v60,z5,tPen\WObj:=wPaper;
    MoveL Offs(pOrigin,237.46,260.21,6.00),vTravel,z5,tPen\WObj:=wPaper;
    MoveL Offs(pOrigin,237.46,260.21,0.00),v60,z0,tPen\WObj:=wPaper;
    MoveL Offs(pOrigin,237.04,260.42,0.00),v40,z0,tPen\WObj:=wPaper;
    MoveL Offs(pOrigin,237.04,261.49,0.00),v40,z0,tPen\WObj:=wPaper;
    MoveL Offs(pOrigin,237.68,262.12,0.00),v40,fine,tPen\WObj:=wPaper;
    MoveL Offs(pOrigin,237.68,262.12,6.00),v60,z5,tPen\WObj:=wPaper;
    MoveL Offs(pOrigin,235.76,261.06,6.00),vTravel,z5,tPen\WObj:=wPaper;
    MoveL Offs(pOrigin,235.76,261.06,0.00),v60,z0,tPen\WObj:=wPaper;
    MoveL Offs(pOrigin,235.76,259.58,0.00),v40,z0,tPen\WObj:=wPaper;
    MoveL Offs(pOrigin,235.34,259.36,0.00),v40,z0,tPen\WObj:=wPaper;
    MoveL Offs(pOrigin,235.34,259.36,0.00),v40,z0,tPen\WObj:=wPaper;
    MoveL Offs(pOrigin,235.34,257.88,0.00),v40,fine,tPen\WObj:=wPaper;
    MoveL Offs(pOrigin,235.34,257.88,6.00),v60,z5,tPen\WObj:=wPaper;
    MoveL Offs(pOrigin,235.34,259.36,6.00),vTravel,z5,tPen\WObj:=wPaper;
    MoveL Offs(pOrigin,235.34,259.36,0.00),v60,z0,tPen\WObj:=wPaper;
    MoveL Offs(pOrigin,234.70,260.00,0.00),v40,z0,tPen\WObj:=wPaper;
    MoveL Offs(pOrigin,234.70,260.00,0.00),v40,z0,tPen\WObj:=wPaper;
    MoveL Offs(pOrigin,235.69,261.27,0.00),v40,z0,tPen\WObj:=wPaper;
    MoveL Offs(pOrigin,235.98,262.34,0.00),v40,z0,tPen\WObj:=wPaper;
    MoveL Offs(pOrigin,235.34,264.25,0.00),v40,z0,tPen\WObj:=wPaper;
    MoveL Offs(pOrigin,235.34,264.46,0.00),v40,z0,tPen\WObj:=wPaper;
    MoveL Offs(pOrigin,234.06,264.25,0.00),v40,z0,tPen\WObj:=wPaper;
    MoveL Offs(pOrigin,230.02,266.16,0.00),v40,z0,tPen\WObj:=wPaper;
    MoveL Offs(pOrigin,225.14,265.95,0.00),v40,z0,tPen\WObj:=wPaper;
    MoveL Offs(pOrigin,221.52,264.75,0.00),v40,z0,tPen\WObj:=wPaper;
    MoveL Offs(pOrigin,219.82,263.83,0.00),v40,z0,tPen\WObj:=wPaper;
    MoveL Offs(pOrigin,218.12,262.34,0.00),v40,z0,tPen\WObj:=wPaper;
    MoveL Offs(pOrigin,217.49,260.42,0.00),v40,z0,tPen\WObj:=wPaper;
    MoveL Offs(pOrigin,217.49,260.42,0.00),v40,z0,tPen\WObj:=wPaper;
    MoveL Offs(pOrigin,217.06,259.58,0.00),v40,z0,tPen\WObj:=wPaper;
    MoveL Offs(pOrigin,216.21,259.08,0.00),v40,z0,tPen\WObj:=wPaper;
    MoveL Offs(pOrigin,214.30,258.51,0.00),v40,z0,tPen\WObj:=wPaper;
    MoveL Offs(pOrigin,212.81,258.51,0.00),v40,fine,tPen\WObj:=wPaper;
    MoveL Offs(pOrigin,212.81,258.51,6.00),v60,z5,tPen\WObj:=wPaper;
    MoveL Offs(pOrigin,215.36,259.79,6.00),vTravel,z5,tPen\WObj:=wPaper;
    MoveL Offs(pOrigin,215.36,259.79,0.00),v60,z0,tPen\WObj:=wPaper;
    MoveL Offs(pOrigin,217.06,260.64,0.00),v40,z0,tPen\WObj:=wPaper;
    MoveL Offs(pOrigin,217.49,260.42,0.00),v40,z0,tPen\WObj:=wPaper;
    MoveL Offs(pOrigin,220.04,261.27,0.00),v40,z0,tPen\WObj:=wPaper;
    MoveL Offs(pOrigin,220.04,261.27,0.00),v40,z0,tPen\WObj:=wPaper;
    MoveL Offs(pOrigin,220.25,262.12,0.00),v40,z0,tPen\WObj:=wPaper;
    MoveL Offs(pOrigin,222.16,263.54,0.00),v40,z0,tPen\WObj:=wPaper;
    MoveL Offs(pOrigin,223.65,263.61,0.00),v40,z0,tPen\WObj:=wPaper;
    MoveL Offs(pOrigin,223.65,263.61,0.00),v40,z0,tPen\WObj:=wPaper;
    MoveL Offs(pOrigin,223.93,262.55,0.00),v40,z0,tPen\WObj:=wPaper;
    MoveL Offs(pOrigin,225.35,261.70,0.00),v40,z0,tPen\WObj:=wPaper;
    MoveL Offs(pOrigin,225.35,261.70,0.00),v40,z0,tPen\WObj:=wPaper;
    MoveL Offs(pOrigin,223.86,260.21,0.00),v40,z0,tPen\WObj:=wPaper;
    MoveL Offs(pOrigin,220.68,260.85,0.00),v40,z0,tPen\WObj:=wPaper;
    MoveL Offs(pOrigin,220.04,261.27,0.00),v40,fine,tPen\WObj:=wPaper;
    MoveL Offs(pOrigin,220.04,261.27,6.00),v60,z5,tPen\WObj:=wPaper;
    MoveL Offs(pOrigin,223.65,263.61,6.00),vTravel,z5,tPen\WObj:=wPaper;
    MoveL Offs(pOrigin,223.65,263.61,0.00),v60,z0,tPen\WObj:=wPaper;
    MoveL Offs(pOrigin,224.93,264.46,0.00),v40,z0,tPen\WObj:=wPaper;
    MoveL Offs(pOrigin,226.41,264.25,0.00),v40,z0,tPen\WObj:=wPaper;
    MoveL Offs(pOrigin,226.41,264.25,0.00),v40,z0,tPen\WObj:=wPaper;
    MoveL Offs(pOrigin,226.34,262.12,0.00),v40,z0,tPen\WObj:=wPaper;
    MoveL Offs(pOrigin,225.35,261.70,0.00),v40,z0,tPen\WObj:=wPaper;
    MoveL Offs(pOrigin,226.41,261.91,0.00),v40,z0,tPen\WObj:=wPaper;
    MoveL Offs(pOrigin,227.69,262.12,0.00),v40,z0,tPen\WObj:=wPaper;
    MoveL Offs(pOrigin,227.69,262.12,0.00),v40,z0,tPen\WObj:=wPaper;
    MoveL Offs(pOrigin,228.54,262.98,0.00),v40,z0,tPen\WObj:=wPaper;
    MoveL Offs(pOrigin,228.54,264.25,0.00),v40,z0,tPen\WObj:=wPaper;
    MoveL Offs(pOrigin,228.54,264.25,0.00),v40,z0,tPen\WObj:=wPaper;
    MoveL Offs(pOrigin,230.02,264.11,0.00),v40,z0,tPen\WObj:=wPaper;
    MoveL Offs(pOrigin,231.94,263.26,0.00),v40,z0,tPen\WObj:=wPaper;
    MoveL Offs(pOrigin,232.36,262.76,0.00),v40,z0,tPen\WObj:=wPaper;
    MoveL Offs(pOrigin,232.36,262.76,0.00),v40,z0,tPen\WObj:=wPaper;
    MoveL Offs(pOrigin,231.94,261.84,0.00),v40,z0,tPen\WObj:=wPaper;
    MoveL Offs(pOrigin,228.96,261.06,0.00),v40,z0,tPen\WObj:=wPaper;
    MoveL Offs(pOrigin,228.32,261.27,0.00),v40,z0,tPen\WObj:=wPaper;
    MoveL Offs(pOrigin,227.69,262.12,0.00),v40,fine,tPen\WObj:=wPaper;
    MoveL Offs(pOrigin,227.69,262.12,6.00),v60,z5,tPen\WObj:=wPaper;
    MoveL Offs(pOrigin,228.54,264.25,6.00),vTravel,z5,tPen\WObj:=wPaper;
    MoveL Offs(pOrigin,228.54,264.25,0.00),v60,z0,tPen\WObj:=wPaper;
    MoveL Offs(pOrigin,228.11,264.46,0.00),v40,z0,tPen\WObj:=wPaper;
    MoveL Offs(pOrigin,226.41,264.25,0.00),v40,fine,tPen\WObj:=wPaper;
    MoveL Offs(pOrigin,226.41,264.25,6.00),v60,z5,tPen\WObj:=wPaper;
    MoveL Offs(pOrigin,224.29,260.21,6.00),vTravel,z5,tPen\WObj:=wPaper;
    MoveL Offs(pOrigin,224.29,260.21,0.00),v60,z0,tPen\WObj:=wPaper;
    MoveL Offs(pOrigin,224.93,260.85,0.00),v40,z0,tPen\WObj:=wPaper;
    MoveL Offs(pOrigin,224.29,260.21,0.00),v40,fine,tPen\WObj:=wPaper;
    MoveL Offs(pOrigin,224.29,260.21,6.00),v60,z5,tPen\WObj:=wPaper;
    MoveL Offs(pOrigin,223.86,256.60,6.00),vTravel,z5,tPen\WObj:=wPaper;
    MoveL Offs(pOrigin,223.86,256.60,0.00),v60,z0,tPen\WObj:=wPaper;
    MoveL Offs(pOrigin,226.41,257.02,0.00),v40,z0,tPen\WObj:=wPaper;
    MoveL Offs(pOrigin,231.09,259.01,0.00),v40,z0,tPen\WObj:=wPaper;
    MoveL Offs(pOrigin,232.79,259.36,0.00),v40,fine,tPen\WObj:=wPaper;
    MoveL Offs(pOrigin,232.79,259.36,6.00),v60,z5,tPen\WObj:=wPaper;
    MoveL Offs(pOrigin,234.70,260.00,6.00),vTravel,z5,tPen\WObj:=wPaper;
    MoveL Offs(pOrigin,234.70,260.00,0.00),v60,z0,tPen\WObj:=wPaper;
    MoveL Offs(pOrigin,231.30,256.60,0.00),v40,z0,tPen\WObj:=wPaper;
    MoveL Offs(pOrigin,228.96,255.11,0.00),v40,fine,tPen\WObj:=wPaper;
    MoveL Offs(pOrigin,228.96,255.11,6.00),v60,z5,tPen\WObj:=wPaper;
    MoveL Offs(pOrigin,232.36,261.91,6.00),vTravel,z5,tPen\WObj:=wPaper;
    MoveL Offs(pOrigin,232.36,261.91,0.00),v60,z0,tPen\WObj:=wPaper;
  ENDPROC

  PROC DrawPart7()
    MoveL Offs(pOrigin,233.85,261.70,0.00),v40,z0,tPen\WObj:=wPaper;
    MoveL Offs(pOrigin,234.06,262.34,0.00),v40,z0,tPen\WObj:=wPaper;
    MoveL Offs(pOrigin,232.36,262.76,0.00),v40,fine,tPen\WObj:=wPaper;
    MoveL Offs(pOrigin,232.36,262.76,6.00),v60,z5,tPen\WObj:=wPaper;
    MoveL Offs(pOrigin,235.34,264.46,6.00),vTravel,z5,tPen\WObj:=wPaper;
    MoveL Offs(pOrigin,235.34,264.46,0.00),v60,z0,tPen\WObj:=wPaper;
    MoveL Offs(pOrigin,235.55,265.52,0.00),v40,z0,tPen\WObj:=wPaper;
    MoveL Offs(pOrigin,235.20,266.38,0.00),v40,z0,tPen\WObj:=wPaper;
    MoveL Offs(pOrigin,233.64,267.72,0.00),v40,z0,tPen\WObj:=wPaper;
    MoveL Offs(pOrigin,230.88,268.29,0.00),v40,z0,tPen\WObj:=wPaper;
    MoveL Offs(pOrigin,225.14,268.08,0.00),v40,z0,tPen\WObj:=wPaper;
    MoveL Offs(pOrigin,223.44,267.65,0.00),v40,z0,tPen\WObj:=wPaper;
    MoveL Offs(pOrigin,219.40,267.44,0.00),v40,z0,tPen\WObj:=wPaper;
    MoveL Offs(pOrigin,215.57,266.23,0.00),v40,z0,tPen\WObj:=wPaper;
    MoveL Offs(pOrigin,214.73,265.74,0.00),v40,z0,tPen\WObj:=wPaper;
    MoveL Offs(pOrigin,213.45,264.25,0.00),v40,z0,tPen\WObj:=wPaper;
    MoveL Offs(pOrigin,213.02,262.76,0.00),v40,fine,tPen\WObj:=wPaper;
    MoveL Offs(pOrigin,213.02,262.76,6.00),v60,z5,tPen\WObj:=wPaper;
    MoveL Offs(pOrigin,208.14,265.31,6.00),vTravel,z5,tPen\WObj:=wPaper;
    MoveL Offs(pOrigin,208.14,265.31,0.00),v60,z0,tPen\WObj:=wPaper;
    MoveL Offs(pOrigin,205.80,264.67,0.00),v40,z0,tPen\WObj:=wPaper;
    MoveL Offs(pOrigin,204.74,265.52,0.00),v40,z0,tPen\WObj:=wPaper;
    MoveL Offs(pOrigin,204.74,265.52,0.00),v40,z0,tPen\WObj:=wPaper;
    MoveL Offs(pOrigin,204.95,271.05,0.00),v40,z0,tPen\WObj:=wPaper;
    MoveL Offs(pOrigin,205.38,271.90,0.00),v40,z0,tPen\WObj:=wPaper;
    MoveL Offs(pOrigin,205.38,273.39,0.00),v40,fine,tPen\WObj:=wPaper;
    MoveL Offs(pOrigin,205.38,273.39,6.00),v60,z5,tPen\WObj:=wPaper;
    MoveL Offs(pOrigin,203.89,273.81,6.00),vTravel,z5,tPen\WObj:=wPaper;
    MoveL Offs(pOrigin,203.89,273.81,0.00),v60,z0,tPen\WObj:=wPaper;
    MoveL Offs(pOrigin,203.60,272.11,0.00),v40,z0,tPen\WObj:=wPaper;
    MoveL Offs(pOrigin,202.68,271.26,0.00),v40,z0,tPen\WObj:=wPaper;
    MoveL Offs(pOrigin,202.12,268.92,0.00),v40,z0,tPen\WObj:=wPaper;
    MoveL Offs(pOrigin,199.85,267.65,0.00),v40,z0,tPen\WObj:=wPaper;
    MoveL Offs(pOrigin,199.85,267.65,0.00),v40,z0,tPen\WObj:=wPaper;
    MoveL Offs(pOrigin,199.85,266.16,0.00),v40,z0,tPen\WObj:=wPaper;
    MoveL Offs(pOrigin,200.27,265.95,0.00),v40,z0,tPen\WObj:=wPaper;
    MoveL Offs(pOrigin,200.27,265.95,0.00),v40,z0,tPen\WObj:=wPaper;
    MoveL Offs(pOrigin,200.06,264.46,0.00),v40,z0,tPen\WObj:=wPaper;
    MoveL Offs(pOrigin,197.73,263.19,0.00),v40,z0,tPen\WObj:=wPaper;
    MoveL Offs(pOrigin,196.17,261.06,0.00),v40,z0,tPen\WObj:=wPaper;
    MoveL Offs(pOrigin,195.39,257.45,0.00),v40,z0,tPen\WObj:=wPaper;
    MoveL Offs(pOrigin,195.39,255.11,0.00),v40,z0,tPen\WObj:=wPaper;
    MoveL Offs(pOrigin,196.73,250.65,0.00),v40,z0,tPen\WObj:=wPaper;
    MoveL Offs(pOrigin,200.35,244.70,0.00),v40,z0,tPen\WObj:=wPaper;
    MoveL Offs(pOrigin,201.34,241.94,0.00),v40,z0,tPen\WObj:=wPaper;
    MoveL Offs(pOrigin,201.76,239.60,0.00),v40,z0,tPen\WObj:=wPaper;
    MoveL Offs(pOrigin,201.76,239.60,0.00),v40,z0,tPen\WObj:=wPaper;
    MoveL Offs(pOrigin,186.04,236.84,0.00),v40,z0,tPen\WObj:=wPaper;
    MoveL Offs(pOrigin,178.60,234.78,0.00),v40,z0,tPen\WObj:=wPaper;
    MoveL Offs(pOrigin,175.20,233.51,0.00),v40,z0,tPen\WObj:=wPaper;
    MoveL Offs(pOrigin,170.74,231.17,0.00),v40,z0,tPen\WObj:=wPaper;
    MoveL Offs(pOrigin,167.98,229.19,0.00),v40,z0,tPen\WObj:=wPaper;
    MoveL Offs(pOrigin,165.85,227.06,0.00),v40,z0,tPen\WObj:=wPaper;
    MoveL Offs(pOrigin,162.80,222.18,0.00),v40,z0,tPen\WObj:=wPaper;
    MoveL Offs(pOrigin,161.18,216.65,0.00),v40,z0,tPen\WObj:=wPaper;
    MoveL Offs(pOrigin,160.32,206.66,0.00),v40,z0,tPen\WObj:=wPaper;
    MoveL Offs(pOrigin,160.32,193.27,0.00),v40,z0,tPen\WObj:=wPaper;
    MoveL Offs(pOrigin,160.32,193.27,0.00),v40,z0,tPen\WObj:=wPaper;
    MoveL Offs(pOrigin,161.39,193.27,0.00),v40,z0,tPen\WObj:=wPaper;
    MoveL Offs(pOrigin,166.70,194.83,0.00),v40,z0,tPen\WObj:=wPaper;
    MoveL Offs(pOrigin,167.34,195.40,0.00),v40,fine,tPen\WObj:=wPaper;
    MoveL Offs(pOrigin,167.34,195.40,6.00),v60,z5,tPen\WObj:=wPaper;
    MoveL Offs(pOrigin,160.32,193.27,6.00),vTravel,z5,tPen\WObj:=wPaper;
    MoveL Offs(pOrigin,160.32,193.27,0.00),v60,z0,tPen\WObj:=wPaper;
    MoveL Offs(pOrigin,159.69,192.57,0.00),v40,z0,tPen\WObj:=wPaper;
    MoveL Offs(pOrigin,150.12,189.88,0.00),v40,z0,tPen\WObj:=wPaper;
    MoveL Offs(pOrigin,145.45,188.25,0.00),v40,z0,tPen\WObj:=wPaper;
    MoveL Offs(pOrigin,145.02,187.75,0.00),v40,z0,tPen\WObj:=wPaper;
    MoveL Offs(pOrigin,145.02,187.75,0.00),v40,z0,tPen\WObj:=wPaper;
    MoveL Offs(pOrigin,143.54,187.61,0.00),v40,z0,tPen\WObj:=wPaper;
    MoveL Offs(pOrigin,142.05,186.69,0.00),v40,z0,tPen\WObj:=wPaper;
    MoveL Offs(pOrigin,140.77,185.41,0.00),v40,z0,tPen\WObj:=wPaper;
    MoveL Offs(pOrigin,139.00,182.44,0.00),v40,z0,tPen\WObj:=wPaper;
    MoveL Offs(pOrigin,138.01,179.25,0.00),v40,z0,tPen\WObj:=wPaper;
    MoveL Offs(pOrigin,136.95,173.30,0.00),v40,z0,tPen\WObj:=wPaper;
    MoveL Offs(pOrigin,135.68,170.11,0.00),v40,z0,tPen\WObj:=wPaper;
    MoveL Offs(pOrigin,135.18,167.77,0.00),v40,z0,tPen\WObj:=wPaper;
    MoveL Offs(pOrigin,134.33,167.14,0.00),v40,z0,tPen\WObj:=wPaper;
    MoveL Offs(pOrigin,133.76,165.86,0.00),v40,z0,tPen\WObj:=wPaper;
    MoveL Offs(pOrigin,133.55,160.98,0.00),v40,z0,tPen\WObj:=wPaper;
    MoveL Offs(pOrigin,133.12,160.12,0.00),v40,z0,tPen\WObj:=wPaper;
    MoveL Offs(pOrigin,131.00,158.21,0.00),v40,z0,tPen\WObj:=wPaper;
    MoveL Offs(pOrigin,130.50,157.36,0.00),v40,z0,tPen\WObj:=wPaper;
    MoveL Offs(pOrigin,130.15,155.45,0.00),v40,z0,tPen\WObj:=wPaper;
    MoveL Offs(pOrigin,130.36,152.05,0.00),v40,z0,tPen\WObj:=wPaper;
    MoveL Offs(pOrigin,129.80,150.35,0.00),v40,z0,tPen\WObj:=wPaper;
    MoveL Offs(pOrigin,127.32,147.38,0.00),v40,z0,tPen\WObj:=wPaper;
    MoveL Offs(pOrigin,126.82,144.82,0.00),v40,z0,tPen\WObj:=wPaper;
    MoveL Offs(pOrigin,126.96,140.57,0.00),v40,z0,tPen\WObj:=wPaper;
    MoveL Offs(pOrigin,126.18,138.88,0.00),v40,z0,tPen\WObj:=wPaper;
    MoveL Offs(pOrigin,124.06,136.11,0.00),v40,z0,tPen\WObj:=wPaper;
    MoveL Offs(pOrigin,123.78,133.14,0.00),v40,z0,tPen\WObj:=wPaper;
    MoveL Offs(pOrigin,123.78,133.14,0.00),v40,z0,tPen\WObj:=wPaper;
    MoveL Offs(pOrigin,121.01,132.57,0.00),v40,z0,tPen\WObj:=wPaper;
    MoveL Offs(pOrigin,119.95,131.86,0.00),v40,z0,tPen\WObj:=wPaper;
    MoveL Offs(pOrigin,118.82,130.38,0.00),v40,z0,tPen\WObj:=wPaper;
    MoveL Offs(pOrigin,117.40,122.72,0.00),v40,z0,tPen\WObj:=wPaper;
    MoveL Offs(pOrigin,116.20,118.90,0.00),v40,z0,tPen\WObj:=wPaper;
    MoveL Offs(pOrigin,114.21,115.71,0.00),v40,z0,tPen\WObj:=wPaper;
    MoveL Offs(pOrigin,110.81,111.89,0.00),v40,z0,tPen\WObj:=wPaper;
    MoveL Offs(pOrigin,108.19,108.06,0.00),v40,z0,tPen\WObj:=wPaper;
    MoveL Offs(pOrigin,105.71,101.69,0.00),v40,z0,tPen\WObj:=wPaper;
    MoveL Offs(pOrigin,104.22,96.59,0.00),v40,z0,tPen\WObj:=wPaper;
    MoveL Offs(pOrigin,104.01,94.68,0.00),v40,z0,tPen\WObj:=wPaper;
    MoveL Offs(pOrigin,104.01,94.68,0.00),v40,z0,tPen\WObj:=wPaper;
    MoveL Offs(pOrigin,106.14,95.24,0.00),v40,z0,tPen\WObj:=wPaper;
    MoveL Offs(pOrigin,116.12,101.33,0.00),v40,z0,tPen\WObj:=wPaper;
    MoveL Offs(pOrigin,119.10,102.75,0.00),v40,fine,tPen\WObj:=wPaper;
    MoveL Offs(pOrigin,119.10,102.75,6.00),v60,z5,tPen\WObj:=wPaper;
    MoveL Offs(pOrigin,112.09,107.00,6.00),vTravel,z5,tPen\WObj:=wPaper;
    MoveL Offs(pOrigin,112.09,107.00,0.00),v60,z0,tPen\WObj:=wPaper;
    MoveL Offs(pOrigin,112.94,107.85,0.00),v40,z0,tPen\WObj:=wPaper;
    MoveL Offs(pOrigin,112.09,107.00,0.00),v40,fine,tPen\WObj:=wPaper;
    MoveL Offs(pOrigin,112.09,107.00,6.00),v60,z5,tPen\WObj:=wPaper;
    MoveL Offs(pOrigin,108.26,107.85,6.00),vTravel,z5,tPen\WObj:=wPaper;
    MoveL Offs(pOrigin,108.26,107.85,0.00),v60,z0,tPen\WObj:=wPaper;
    MoveL Offs(pOrigin,108.47,108.28,0.00),v40,z0,tPen\WObj:=wPaper;
    MoveL Offs(pOrigin,108.26,107.85,0.00),v40,z0,tPen\WObj:=wPaper;
    MoveL Offs(pOrigin,107.84,107.00,0.00),v40,z0,tPen\WObj:=wPaper;
    MoveL Offs(pOrigin,108.05,107.43,0.00),v40,z0,tPen\WObj:=wPaper;
  ENDPROC

  PROC DrawPart8()
    MoveL Offs(pOrigin,107.84,107.00,0.00),v40,fine,tPen\WObj:=wPaper;
    MoveL Offs(pOrigin,107.84,107.00,6.00),v60,z5,tPen\WObj:=wPaper;
    MoveL Offs(pOrigin,106.78,104.45,6.00),vTravel,z5,tPen\WObj:=wPaper;
    MoveL Offs(pOrigin,106.78,104.45,0.00),v60,z0,tPen\WObj:=wPaper;
    MoveL Offs(pOrigin,106.99,104.88,0.00),v40,z0,tPen\WObj:=wPaper;
    MoveL Offs(pOrigin,106.78,104.45,0.00),v40,fine,tPen\WObj:=wPaper;
    MoveL Offs(pOrigin,106.78,104.45,6.00),v60,z5,tPen\WObj:=wPaper;
    MoveL Offs(pOrigin,108.05,100.62,6.00),vTravel,z5,tPen\WObj:=wPaper;
    MoveL Offs(pOrigin,108.05,100.62,0.00),v60,z0,tPen\WObj:=wPaper;
    MoveL Offs(pOrigin,108.26,101.05,0.00),v40,z0,tPen\WObj:=wPaper;
    MoveL Offs(pOrigin,108.05,100.62,0.00),v40,fine,tPen\WObj:=wPaper;
    MoveL Offs(pOrigin,108.05,100.62,6.00),v60,z5,tPen\WObj:=wPaper;
    MoveL Offs(pOrigin,107.20,98.93,6.00),vTravel,z5,tPen\WObj:=wPaper;
    MoveL Offs(pOrigin,107.20,98.93,0.00),v60,z0,tPen\WObj:=wPaper;
    MoveL Offs(pOrigin,108.40,101.69,0.00),v40,z0,tPen\WObj:=wPaper;
    MoveL Offs(pOrigin,112.09,107.21,0.00),v40,z0,tPen\WObj:=wPaper;
    MoveL Offs(pOrigin,114.43,109.34,0.00),v40,z0,tPen\WObj:=wPaper;
    MoveL Offs(pOrigin,119.31,112.17,0.00),v40,z0,tPen\WObj:=wPaper;
    MoveL Offs(pOrigin,123.78,113.80,0.00),v40,z0,tPen\WObj:=wPaper;
    MoveL Offs(pOrigin,126.96,114.44,0.00),v40,fine,tPen\WObj:=wPaper;
    MoveL Offs(pOrigin,126.96,114.44,6.00),v60,z5,tPen\WObj:=wPaper;
    MoveL Offs(pOrigin,125.90,111.25,6.00),vTravel,z5,tPen\WObj:=wPaper;
    MoveL Offs(pOrigin,125.90,111.25,0.00),v60,z0,tPen\WObj:=wPaper;
    MoveL Offs(pOrigin,131.43,112.10,0.00),v40,z0,tPen\WObj:=wPaper;
    MoveL Offs(pOrigin,141.62,112.31,0.00),v40,z0,tPen\WObj:=wPaper;
    MoveL Offs(pOrigin,156.07,110.82,0.00),v40,z0,tPen\WObj:=wPaper;
    MoveL Offs(pOrigin,161.81,110.82,0.00),v40,fine,tPen\WObj:=wPaper;
    MoveL Offs(pOrigin,161.81,110.82,6.00),v60,z5,tPen\WObj:=wPaper;
    MoveL Offs(pOrigin,162.66,108.28,6.00),vTravel,z5,tPen\WObj:=wPaper;
    MoveL Offs(pOrigin,162.66,108.28,0.00),v60,z0,tPen\WObj:=wPaper;
    MoveL Offs(pOrigin,162.24,108.91,0.00),v40,z0,tPen\WObj:=wPaper;
    MoveL Offs(pOrigin,161.81,112.31,0.00),v40,z0,tPen\WObj:=wPaper;
    MoveL Offs(pOrigin,161.18,114.44,0.00),v40,z0,tPen\WObj:=wPaper;
    MoveL Offs(pOrigin,161.18,114.44,0.00),v40,z0,tPen\WObj:=wPaper;
    MoveL Offs(pOrigin,161.39,115.07,0.00),v40,z0,tPen\WObj:=wPaper;
    MoveL Offs(pOrigin,159.90,124.00,0.00),v40,z0,tPen\WObj:=wPaper;
    MoveL Offs(pOrigin,159.90,124.00,0.00),v40,z0,tPen\WObj:=wPaper;
    MoveL Offs(pOrigin,159.69,126.76,0.00),v40,z0,tPen\WObj:=wPaper;
    MoveL Offs(pOrigin,159.05,128.46,0.00),v40,z0,tPen\WObj:=wPaper;
    MoveL Offs(pOrigin,159.05,128.46,0.00),v40,z0,tPen\WObj:=wPaper;
    MoveL Offs(pOrigin,159.05,129.95,0.00),v40,z0,tPen\WObj:=wPaper;
    MoveL Offs(pOrigin,158.41,132.71,0.00),v40,z0,tPen\WObj:=wPaper;
    MoveL Offs(pOrigin,157.14,135.48,0.00),v40,fine,tPen\WObj:=wPaper;
    MoveL Offs(pOrigin,157.14,135.48,6.00),v60,z5,tPen\WObj:=wPaper;
    MoveL Offs(pOrigin,155.65,135.69,6.00),vTravel,z5,tPen\WObj:=wPaper;
    MoveL Offs(pOrigin,155.65,135.69,0.00),v60,z0,tPen\WObj:=wPaper;
    MoveL Offs(pOrigin,154.94,137.60,0.00),v40,z0,tPen\WObj:=wPaper;
    MoveL Offs(pOrigin,148.35,145.25,0.00),v40,z0,tPen\WObj:=wPaper;
    MoveL Offs(pOrigin,140.99,152.05,0.00),v40,z0,tPen\WObj:=wPaper;
    MoveL Offs(pOrigin,140.56,152.26,0.00),v40,z0,tPen\WObj:=wPaper;
    MoveL Offs(pOrigin,136.10,154.88,0.00),v40,z0,tPen\WObj:=wPaper;
    MoveL Offs(pOrigin,135.04,155.02,0.00),v40,fine,tPen\WObj:=wPaper;
    MoveL Offs(pOrigin,135.04,155.02,6.00),v60,z5,tPen\WObj:=wPaper;
    MoveL Offs(pOrigin,140.77,159.49,6.00),vTravel,z5,tPen\WObj:=wPaper;
    MoveL Offs(pOrigin,140.77,159.49,0.00),v60,z0,tPen\WObj:=wPaper;
    MoveL Offs(pOrigin,140.99,159.06,0.00),v40,z0,tPen\WObj:=wPaper;
    MoveL Offs(pOrigin,140.77,159.49,0.00),v40,z0,tPen\WObj:=wPaper;
    MoveL Offs(pOrigin,140.14,160.34,0.00),v40,z0,tPen\WObj:=wPaper;
    MoveL Offs(pOrigin,140.35,159.91,0.00),v40,z0,tPen\WObj:=wPaper;
    MoveL Offs(pOrigin,140.14,160.34,0.00),v40,fine,tPen\WObj:=wPaper;
    MoveL Offs(pOrigin,140.14,160.34,6.00),v60,z5,tPen\WObj:=wPaper;
    MoveL Offs(pOrigin,139.29,161.19,6.00),vTravel,z5,tPen\WObj:=wPaper;
    MoveL Offs(pOrigin,139.29,161.19,0.00),v60,z0,tPen\WObj:=wPaper;
    MoveL Offs(pOrigin,139.07,161.61,0.00),v40,z0,tPen\WObj:=wPaper;
    MoveL Offs(pOrigin,139.29,161.19,0.00),v40,fine,tPen\WObj:=wPaper;
    MoveL Offs(pOrigin,139.29,161.19,6.00),v60,z5,tPen\WObj:=wPaper;
    MoveL Offs(pOrigin,141.62,158.43,6.00),vTravel,z5,tPen\WObj:=wPaper;
    MoveL Offs(pOrigin,141.62,158.43,0.00),v60,z0,tPen\WObj:=wPaper;
    MoveL Offs(pOrigin,141.41,158.85,0.00),v40,z0,tPen\WObj:=wPaper;
    MoveL Offs(pOrigin,141.62,158.43,0.00),v40,fine,tPen\WObj:=wPaper;
    MoveL Offs(pOrigin,141.62,158.43,6.00),v60,z5,tPen\WObj:=wPaper;
    MoveL Offs(pOrigin,144.39,155.45,6.00),vTravel,z5,tPen\WObj:=wPaper;
    MoveL Offs(pOrigin,144.39,155.45,0.00),v60,z0,tPen\WObj:=wPaper;
    MoveL Offs(pOrigin,144.18,155.88,0.00),v40,z0,tPen\WObj:=wPaper;
    MoveL Offs(pOrigin,144.39,155.45,0.00),v40,z0,tPen\WObj:=wPaper;
    MoveL Offs(pOrigin,145.02,154.81,0.00),v40,z0,tPen\WObj:=wPaper;
    MoveL Offs(pOrigin,144.81,155.24,0.00),v40,z0,tPen\WObj:=wPaper;
    MoveL Offs(pOrigin,145.02,154.81,0.00),v40,fine,tPen\WObj:=wPaper;
    MoveL Offs(pOrigin,145.02,154.81,6.00),v60,z5,tPen\WObj:=wPaper;
    MoveL Offs(pOrigin,147.36,152.69,6.00),vTravel,z5,tPen\WObj:=wPaper;
    MoveL Offs(pOrigin,147.36,152.69,0.00),v60,z0,tPen\WObj:=wPaper;
    MoveL Offs(pOrigin,147.15,153.11,0.00),v40,z0,tPen\WObj:=wPaper;
    MoveL Offs(pOrigin,147.36,152.69,0.00),v40,z0,tPen\WObj:=wPaper;
    MoveL Offs(pOrigin,148.00,152.05,0.00),v40,z0,tPen\WObj:=wPaper;
    MoveL Offs(pOrigin,147.79,152.48,0.00),v40,z0,tPen\WObj:=wPaper;
    MoveL Offs(pOrigin,148.00,152.05,0.00),v40,fine,tPen\WObj:=wPaper;
    MoveL Offs(pOrigin,148.00,152.05,6.00),v60,z5,tPen\WObj:=wPaper;
    MoveL Offs(pOrigin,149.70,150.56,6.00),vTravel,z5,tPen\WObj:=wPaper;
    MoveL Offs(pOrigin,149.70,150.56,0.00),v60,z0,tPen\WObj:=wPaper;
    MoveL Offs(pOrigin,140.63,159.49,0.00),v40,z0,tPen\WObj:=wPaper;
    MoveL Offs(pOrigin,136.88,164.80,0.00),v40,z0,tPen\WObj:=wPaper;
    MoveL Offs(pOrigin,135.68,167.35,0.00),v40,z0,tPen\WObj:=wPaper;
    MoveL Offs(pOrigin,135.25,167.56,0.00),v40,fine,tPen\WObj:=wPaper;
    MoveL Offs(pOrigin,135.25,167.56,6.00),v60,z5,tPen\WObj:=wPaper;
    MoveL Offs(pOrigin,135.89,170.32,6.00),vTravel,z5,tPen\WObj:=wPaper;
    MoveL Offs(pOrigin,135.89,170.32,0.00),v60,z0,tPen\WObj:=wPaper;
    MoveL Offs(pOrigin,136.10,170.75,0.00),v40,z0,tPen\WObj:=wPaper;
    MoveL Offs(pOrigin,135.89,170.32,0.00),v40,fine,tPen\WObj:=wPaper;
    MoveL Offs(pOrigin,135.89,170.32,6.00),v60,z5,tPen\WObj:=wPaper;
    MoveL Offs(pOrigin,143.11,171.60,6.00),vTravel,z5,tPen\WObj:=wPaper;
    MoveL Offs(pOrigin,143.11,171.60,0.00),v60,z0,tPen\WObj:=wPaper;
    MoveL Offs(pOrigin,143.89,169.26,0.00),v40,z0,tPen\WObj:=wPaper;
    MoveL Offs(pOrigin,148.85,159.91,0.00),v40,z0,tPen\WObj:=wPaper;
    MoveL Offs(pOrigin,149.91,159.35,0.00),v40,z0,tPen\WObj:=wPaper;
    MoveL Offs(pOrigin,150.12,160.55,0.00),v40,z0,tPen\WObj:=wPaper;
    MoveL Offs(pOrigin,146.94,170.96,0.00),v40,z0,tPen\WObj:=wPaper;
    MoveL Offs(pOrigin,145.24,178.19,0.00),v40,z0,tPen\WObj:=wPaper;
    MoveL Offs(pOrigin,144.81,180.95,0.00),v40,z0,tPen\WObj:=wPaper;
    MoveL Offs(pOrigin,145.02,187.75,0.00),v40,fine,tPen\WObj:=wPaper;
    MoveL Offs(pOrigin,145.02,187.75,6.00),v60,z5,tPen\WObj:=wPaper;
    MoveL Offs(pOrigin,159.90,190.09,6.00),vTravel,z5,tPen\WObj:=wPaper;
    MoveL Offs(pOrigin,159.90,190.09,0.00),v60,z0,tPen\WObj:=wPaper;
    MoveL Offs(pOrigin,172.44,193.70,0.00),v40,z0,tPen\WObj:=wPaper;
    MoveL Offs(pOrigin,179.45,196.18,0.00),v40,z0,tPen\WObj:=wPaper;
    MoveL Offs(pOrigin,183.49,197.88,0.00),v40,z0,tPen\WObj:=wPaper;
    MoveL Offs(pOrigin,194.32,203.33,0.00),v40,z0,tPen\WObj:=wPaper;
    MoveL Offs(pOrigin,199.00,204.96,0.00),v40,z0,tPen\WObj:=wPaper;
    MoveL Offs(pOrigin,202.82,205.81,0.00),v40,z0,tPen\WObj:=wPaper;
    MoveL Offs(pOrigin,210.69,206.88,0.00),v40,z0,tPen\WObj:=wPaper;
    MoveL Offs(pOrigin,210.69,206.88,0.00),v40,z0,tPen\WObj:=wPaper;
  ENDPROC

  PROC DrawPart9()
    MoveL Offs(pOrigin,212.18,207.73,0.00),v40,z0,tPen\WObj:=wPaper;
    MoveL Offs(pOrigin,215.79,211.34,0.00),v40,z0,tPen\WObj:=wPaper;
    MoveL Offs(pOrigin,216.43,212.82,0.00),v40,z0,tPen\WObj:=wPaper;
    MoveL Offs(pOrigin,216.43,212.82,0.00),v40,z0,tPen\WObj:=wPaper;
    MoveL Offs(pOrigin,214.51,213.04,0.00),v40,z0,tPen\WObj:=wPaper;
    MoveL Offs(pOrigin,208.56,212.19,0.00),v40,z0,tPen\WObj:=wPaper;
    MoveL Offs(pOrigin,201.12,210.13,0.00),v40,z0,tPen\WObj:=wPaper;
    MoveL Offs(pOrigin,197.09,208.43,0.00),v40,z0,tPen\WObj:=wPaper;
    MoveL Offs(pOrigin,180.94,200.22,0.00),v40,z0,tPen\WObj:=wPaper;
    MoveL Offs(pOrigin,173.71,197.31,0.00),v40,z0,tPen\WObj:=wPaper;
    MoveL Offs(pOrigin,172.44,197.10,0.00),v40,z0,tPen\WObj:=wPaper;
    MoveL Offs(pOrigin,172.01,197.31,0.00),v40,z0,tPen\WObj:=wPaper;
    MoveL Offs(pOrigin,170.31,202.62,0.00),v40,z0,tPen\WObj:=wPaper;
    MoveL Offs(pOrigin,168.82,210.91,0.00),v40,z0,tPen\WObj:=wPaper;
    MoveL Offs(pOrigin,168.82,216.86,0.00),v40,z0,tPen\WObj:=wPaper;
    MoveL Offs(pOrigin,169.25,220.05,0.00),v40,z0,tPen\WObj:=wPaper;
    MoveL Offs(pOrigin,170.03,222.81,0.00),v40,z0,tPen\WObj:=wPaper;
    MoveL Offs(pOrigin,172.23,227.06,0.00),v40,z0,tPen\WObj:=wPaper;
    MoveL Offs(pOrigin,175.41,230.25,0.00),v40,z0,tPen\WObj:=wPaper;
    MoveL Offs(pOrigin,180.30,232.87,0.00),v40,z0,tPen\WObj:=wPaper;
    MoveL Offs(pOrigin,184.98,234.29,0.00),v40,z0,tPen\WObj:=wPaper;
    MoveL Offs(pOrigin,186.04,234.29,0.00),v40,fine,tPen\WObj:=wPaper;
    MoveL Offs(pOrigin,186.04,234.29,6.00),v60,z5,tPen\WObj:=wPaper;
    MoveL Offs(pOrigin,177.32,231.52,6.00),vTravel,z5,tPen\WObj:=wPaper;
    MoveL Offs(pOrigin,177.32,231.52,0.00),v60,z0,tPen\WObj:=wPaper;
    MoveL Offs(pOrigin,177.75,231.74,0.00),v40,z0,tPen\WObj:=wPaper;
    MoveL Offs(pOrigin,177.32,231.52,0.00),v40,z0,tPen\WObj:=wPaper;
    MoveL Offs(pOrigin,176.48,231.10,0.00),v40,z0,tPen\WObj:=wPaper;
    MoveL Offs(pOrigin,176.90,231.31,0.00),v40,z0,tPen\WObj:=wPaper;
    MoveL Offs(pOrigin,176.48,231.10,0.00),v40,fine,tPen\WObj:=wPaper;
    MoveL Offs(pOrigin,176.48,231.10,6.00),v60,z5,tPen\WObj:=wPaper;
    MoveL Offs(pOrigin,202.82,233.44,6.00),vTravel,z5,tPen\WObj:=wPaper;
    MoveL Offs(pOrigin,202.82,233.44,0.00),v60,z0,tPen\WObj:=wPaper;
    MoveL Offs(pOrigin,202.61,237.05,0.00),v40,z0,tPen\WObj:=wPaper;
    MoveL Offs(pOrigin,201.76,239.60,0.00),v40,fine,tPen\WObj:=wPaper;
    MoveL Offs(pOrigin,201.76,239.60,6.00),v60,z5,tPen\WObj:=wPaper;
    MoveL Offs(pOrigin,200.70,243.43,6.00),vTravel,z5,tPen\WObj:=wPaper;
    MoveL Offs(pOrigin,200.70,243.43,0.00),v60,z0,tPen\WObj:=wPaper;
    MoveL Offs(pOrigin,200.49,243.85,0.00),v40,z0,tPen\WObj:=wPaper;
    MoveL Offs(pOrigin,200.70,243.43,0.00),v40,z0,tPen\WObj:=wPaper;
    MoveL Offs(pOrigin,200.27,244.49,0.00),v40,z0,tPen\WObj:=wPaper;
    MoveL Offs(pOrigin,200.06,244.91,0.00),v40,z0,tPen\WObj:=wPaper;
    MoveL Offs(pOrigin,200.27,244.49,0.00),v40,fine,tPen\WObj:=wPaper;
    MoveL Offs(pOrigin,200.27,244.49,6.00),v60,z5,tPen\WObj:=wPaper;
    MoveL Offs(pOrigin,205.16,247.89,6.00),vTravel,z5,tPen\WObj:=wPaper;
    MoveL Offs(pOrigin,205.16,247.89,0.00),v60,z0,tPen\WObj:=wPaper;
    MoveL Offs(pOrigin,204.95,244.49,0.00),v40,z0,tPen\WObj:=wPaper;
    MoveL Offs(pOrigin,205.30,243.43,0.00),v40,z0,tPen\WObj:=wPaper;
    MoveL Offs(pOrigin,206.23,242.50,0.00),v40,z0,tPen\WObj:=wPaper;
    MoveL Offs(pOrigin,206.65,243.00,0.00),v40,z0,tPen\WObj:=wPaper;
    MoveL Offs(pOrigin,206.86,247.46,0.00),v40,z0,tPen\WObj:=wPaper;
    MoveL Offs(pOrigin,205.59,253.84,0.00),v40,z0,tPen\WObj:=wPaper;
    MoveL Offs(pOrigin,205.16,257.88,0.00),v40,fine,tPen\WObj:=wPaper;
    MoveL Offs(pOrigin,205.16,257.88,6.00),v60,z5,tPen\WObj:=wPaper;
    MoveL Offs(pOrigin,207.07,259.36,6.00),vTravel,z5,tPen\WObj:=wPaper;
    MoveL Offs(pOrigin,207.07,259.36,0.00),v60,z0,tPen\WObj:=wPaper;
    MoveL Offs(pOrigin,207.64,258.94,0.00),v40,z0,tPen\WObj:=wPaper;
    MoveL Offs(pOrigin,208.92,254.26,0.00),v40,z0,tPen\WObj:=wPaper;
    MoveL Offs(pOrigin,210.90,251.07,0.00),v40,z0,tPen\WObj:=wPaper;
    MoveL Offs(pOrigin,213.45,249.80,0.00),v40,z0,tPen\WObj:=wPaper;
    MoveL Offs(pOrigin,217.06,249.38,0.00),v40,z0,tPen\WObj:=wPaper;
    MoveL Offs(pOrigin,225.56,250.01,0.00),v40,z0,tPen\WObj:=wPaper;
    MoveL Offs(pOrigin,232.15,251.64,0.00),v40,z0,tPen\WObj:=wPaper;
    MoveL Offs(pOrigin,233.85,252.56,0.00),v40,z0,tPen\WObj:=wPaper;
    MoveL Offs(pOrigin,234.91,253.62,0.00),v40,z0,tPen\WObj:=wPaper;
    MoveL Offs(pOrigin,236.61,257.02,0.00),v40,fine,tPen\WObj:=wPaper;
    MoveL Offs(pOrigin,236.61,257.02,6.00),v60,z5,tPen\WObj:=wPaper;
    MoveL Offs(pOrigin,233.21,248.52,6.00),vTravel,z5,tPen\WObj:=wPaper;
    MoveL Offs(pOrigin,233.21,248.52,0.00),v60,z0,tPen\WObj:=wPaper;
    MoveL Offs(pOrigin,231.94,245.34,0.00),v40,z0,tPen\WObj:=wPaper;
    MoveL Offs(pOrigin,232.43,242.86,0.00),v40,z0,tPen\WObj:=wPaper;
    MoveL Offs(pOrigin,233.21,241.94,0.00),v40,z0,tPen\WObj:=wPaper;
    MoveL Offs(pOrigin,234.70,241.30,0.00),v40,z0,tPen\WObj:=wPaper;
    MoveL Offs(pOrigin,236.82,241.94,0.00),v40,z0,tPen\WObj:=wPaper;
    MoveL Offs(pOrigin,239.80,240.80,0.00),v40,z0,tPen\WObj:=wPaper;
    MoveL Offs(pOrigin,240.23,239.81,0.00),v40,z0,tPen\WObj:=wPaper;
    MoveL Offs(pOrigin,240.23,238.75,0.00),v40,z0,tPen\WObj:=wPaper;
    MoveL Offs(pOrigin,239.38,237.26,0.00),v40,z0,tPen\WObj:=wPaper;
    MoveL Offs(pOrigin,239.38,237.26,0.00),v40,z0,tPen\WObj:=wPaper;
    MoveL Offs(pOrigin,240.44,237.33,0.00),v40,z0,tPen\WObj:=wPaper;
    MoveL Offs(pOrigin,242.99,239.39,0.00),v40,z0,tPen\WObj:=wPaper;
    MoveL Offs(pOrigin,244.48,239.39,0.00),v40,z0,tPen\WObj:=wPaper;
    MoveL Offs(pOrigin,246.81,240.24,0.00),v40,z0,tPen\WObj:=wPaper;
    MoveL Offs(pOrigin,246.81,240.24,0.00),v40,z0,tPen\WObj:=wPaper;
    MoveL Offs(pOrigin,246.81,239.81,0.00),v40,z0,tPen\WObj:=wPaper;
    MoveL Offs(pOrigin,247.24,239.81,0.00),v40,z0,tPen\WObj:=wPaper;
    MoveL Offs(pOrigin,247.02,240.24,0.00),v40,z0,tPen\WObj:=wPaper;
    MoveL Offs(pOrigin,247.02,240.24,0.00),v40,z0,tPen\WObj:=wPaper;
    MoveL Offs(pOrigin,247.38,240.24,0.00),v40,z0,tPen\WObj:=wPaper;
    MoveL Offs(pOrigin,247.66,239.39,0.00),v40,z0,tPen\WObj:=wPaper;
    MoveL Offs(pOrigin,248.94,238.11,0.00),v40,z0,tPen\WObj:=wPaper;
    MoveL Offs(pOrigin,248.94,238.11,0.00),v40,z0,tPen\WObj:=wPaper;
    MoveL Offs(pOrigin,248.09,237.26,0.00),v40,z0,tPen\WObj:=wPaper;
    MoveL Offs(pOrigin,248.09,237.26,0.00),v40,z0,tPen\WObj:=wPaper;
    MoveL Offs(pOrigin,248.58,235.14,0.00),v40,z0,tPen\WObj:=wPaper;
    MoveL Offs(pOrigin,249.36,235.00,0.00),v40,z0,tPen\WObj:=wPaper;
    MoveL Offs(pOrigin,251.20,237.05,0.00),v40,z0,tPen\WObj:=wPaper;
    MoveL Offs(pOrigin,251.27,238.32,0.00),v40,z0,tPen\WObj:=wPaper;
    MoveL Offs(pOrigin,251.27,238.32,0.00),v40,z0,tPen\WObj:=wPaper;
    MoveL Offs(pOrigin,251.70,238.75,0.00),v40,z0,tPen\WObj:=wPaper;
    MoveL Offs(pOrigin,253.82,238.54,0.00),v40,z0,tPen\WObj:=wPaper;
    MoveL Offs(pOrigin,253.82,238.54,0.00),v40,z0,tPen\WObj:=wPaper;
    MoveL Offs(pOrigin,253.82,235.77,0.00),v40,z0,tPen\WObj:=wPaper;
    MoveL Offs(pOrigin,253.82,235.77,0.00),v40,z0,tPen\WObj:=wPaper;
    MoveL Offs(pOrigin,254.68,235.35,0.00),v40,z0,tPen\WObj:=wPaper;
    MoveL Offs(pOrigin,255.24,235.56,0.00),v40,z0,tPen\WObj:=wPaper;
    MoveL Offs(pOrigin,255.31,238.32,0.00),v40,z0,tPen\WObj:=wPaper;
    MoveL Offs(pOrigin,255.31,238.32,0.00),v40,z0,tPen\WObj:=wPaper;
    MoveL Offs(pOrigin,258.00,238.54,0.00),v40,z0,tPen\WObj:=wPaper;
    MoveL Offs(pOrigin,258.00,240.02,0.00),v40,z0,tPen\WObj:=wPaper;
    MoveL Offs(pOrigin,257.01,241.51,0.00),v40,fine,tPen\WObj:=wPaper;
    MoveL Offs(pOrigin,257.01,241.51,6.00),v60,z5,tPen\WObj:=wPaper;
    MoveL Offs(pOrigin,258.08,238.32,6.00),vTravel,z5,tPen\WObj:=wPaper;
    MoveL Offs(pOrigin,258.08,238.32,0.00),v60,z0,tPen\WObj:=wPaper;
    MoveL Offs(pOrigin,260.84,238.11,0.00),v40,z0,tPen\WObj:=wPaper;
    MoveL Offs(pOrigin,260.84,238.11,0.00),v40,z0,tPen\WObj:=wPaper;
    MoveL Offs(pOrigin,260.84,239.81,0.00),v40,z0,tPen\WObj:=wPaper;
    MoveL Offs(pOrigin,260.84,239.81,0.00),v40,z0,tPen\WObj:=wPaper;
    MoveL Offs(pOrigin,261.05,240.24,0.00),v40,z0,tPen\WObj:=wPaper;
    MoveL Offs(pOrigin,260.62,240.02,0.00),v40,z0,tPen\WObj:=wPaper;
  ENDPROC

  PROC DrawPart10()
    MoveL Offs(pOrigin,260.84,239.81,0.00),v40,z0,tPen\WObj:=wPaper;
    MoveL Offs(pOrigin,261.05,240.24,0.00),v40,z0,tPen\WObj:=wPaper;
    MoveL Offs(pOrigin,260.62,240.02,0.00),v40,z0,tPen\WObj:=wPaper;
    MoveL Offs(pOrigin,260.84,239.81,0.00),v40,fine,tPen\WObj:=wPaper;
    MoveL Offs(pOrigin,260.84,239.81,6.00),v60,z5,tPen\WObj:=wPaper;
    MoveL Offs(pOrigin,261.48,241.09,6.00),vTravel,z5,tPen\WObj:=wPaper;
    MoveL Offs(pOrigin,261.48,241.09,0.00),v60,z0,tPen\WObj:=wPaper;
    MoveL Offs(pOrigin,261.69,238.54,0.00),v40,z0,tPen\WObj:=wPaper;
    MoveL Offs(pOrigin,261.48,238.18,0.00),v40,z0,tPen\WObj:=wPaper;
    MoveL Offs(pOrigin,260.84,238.11,0.00),v40,z0,tPen\WObj:=wPaper;
    MoveL Offs(pOrigin,261.69,238.11,0.00),v40,z0,tPen\WObj:=wPaper;
    MoveL Offs(pOrigin,262.96,237.69,0.00),v40,z0,tPen\WObj:=wPaper;
    MoveL Offs(pOrigin,262.96,237.69,0.00),v40,z0,tPen\WObj:=wPaper;
    MoveL Offs(pOrigin,262.33,236.84,0.00),v40,z0,tPen\WObj:=wPaper;
    MoveL Offs(pOrigin,262.11,234.29,0.00),v40,fine,tPen\WObj:=wPaper;
    MoveL Offs(pOrigin,262.11,234.29,6.00),v60,z5,tPen\WObj:=wPaper;
    MoveL Offs(pOrigin,263.60,234.50,6.00),vTravel,z5,tPen\WObj:=wPaper;
    MoveL Offs(pOrigin,263.60,234.50,0.00),v60,z0,tPen\WObj:=wPaper;
    MoveL Offs(pOrigin,265.51,236.41,0.00),v40,z0,tPen\WObj:=wPaper;
    MoveL Offs(pOrigin,265.51,236.41,0.00),v40,z0,tPen\WObj:=wPaper;
    MoveL Offs(pOrigin,265.30,237.69,0.00),v40,z0,tPen\WObj:=wPaper;
    MoveL Offs(pOrigin,265.30,237.69,0.00),v40,z0,tPen\WObj:=wPaper;
    MoveL Offs(pOrigin,265.65,237.90,0.00),v40,z0,tPen\WObj:=wPaper;
    MoveL Offs(pOrigin,265.73,239.60,0.00),v40,z0,tPen\WObj:=wPaper;
    MoveL Offs(pOrigin,266.15,240.24,0.00),v40,z0,tPen\WObj:=wPaper;
    MoveL Offs(pOrigin,265.30,240.24,0.00),v40,z0,tPen\WObj:=wPaper;
    MoveL Offs(pOrigin,264.88,240.88,0.00),v40,fine,tPen\WObj:=wPaper;
    MoveL Offs(pOrigin,264.88,240.88,6.00),v60,z5,tPen\WObj:=wPaper;
    MoveL Offs(pOrigin,265.30,237.69,6.00),vTravel,z5,tPen\WObj:=wPaper;
    MoveL Offs(pOrigin,265.30,237.69,0.00),v60,z0,tPen\WObj:=wPaper;
    MoveL Offs(pOrigin,263.39,237.69,0.00),v40,z0,tPen\WObj:=wPaper;
    MoveL Offs(pOrigin,262.54,237.05,0.00),v40,fine,tPen\WObj:=wPaper;
    MoveL Offs(pOrigin,262.54,237.05,6.00),v60,z5,tPen\WObj:=wPaper;
    MoveL Offs(pOrigin,265.51,236.41,6.00),vTravel,z5,tPen\WObj:=wPaper;
    MoveL Offs(pOrigin,265.51,236.41,0.00),v60,z0,tPen\WObj:=wPaper;
    MoveL Offs(pOrigin,263.60,234.36,0.00),v40,z0,tPen\WObj:=wPaper;
    MoveL Offs(pOrigin,260.41,233.65,0.00),v40,z0,tPen\WObj:=wPaper;
    MoveL Offs(pOrigin,254.89,233.44,0.00),v40,z0,tPen\WObj:=wPaper;
    MoveL Offs(pOrigin,245.54,231.74,0.00),v40,z0,tPen\WObj:=wPaper;
    MoveL Offs(pOrigin,239.38,231.52,0.00),v40,z0,tPen\WObj:=wPaper;
    MoveL Offs(pOrigin,235.76,230.68,0.00),v40,z0,tPen\WObj:=wPaper;
    MoveL Offs(pOrigin,233.21,230.68,0.00),v40,fine,tPen\WObj:=wPaper;
    MoveL Offs(pOrigin,233.21,230.68,6.00),v60,z5,tPen\WObj:=wPaper;
    MoveL Offs(pOrigin,234.06,231.52,6.00),vTravel,z5,tPen\WObj:=wPaper;
    MoveL Offs(pOrigin,234.06,231.52,0.00),v60,z0,tPen\WObj:=wPaper;
    MoveL Offs(pOrigin,232.57,230.46,0.00),v40,z0,tPen\WObj:=wPaper;
    MoveL Offs(pOrigin,230.88,230.46,0.00),v40,z0,tPen\WObj:=wPaper;
    MoveL Offs(pOrigin,228.54,232.59,0.00),v40,z0,tPen\WObj:=wPaper;
    MoveL Offs(pOrigin,228.54,232.59,0.00),v40,z0,tPen\WObj:=wPaper;
    MoveL Offs(pOrigin,229.39,233.51,0.00),v40,z0,tPen\WObj:=wPaper;
    MoveL Offs(pOrigin,231.94,234.15,0.00),v40,z0,tPen\WObj:=wPaper;
    MoveL Offs(pOrigin,233.43,235.56,0.00),v40,z0,tPen\WObj:=wPaper;
    MoveL Offs(pOrigin,233.43,235.56,0.00),v40,z0,tPen\WObj:=wPaper;
    MoveL Offs(pOrigin,234.70,235.56,0.00),v40,z0,tPen\WObj:=wPaper;
    MoveL Offs(pOrigin,235.34,236.41,0.00),v40,z0,tPen\WObj:=wPaper;
    MoveL Offs(pOrigin,235.34,236.41,0.00),v40,z0,tPen\WObj:=wPaper;
    MoveL Offs(pOrigin,237.89,236.62,0.00),v40,z0,tPen\WObj:=wPaper;
    MoveL Offs(pOrigin,238.10,236.62,0.00),v40,z0,tPen\WObj:=wPaper;
    MoveL Offs(pOrigin,238.31,237.05,0.00),v40,z0,tPen\WObj:=wPaper;
    MoveL Offs(pOrigin,239.38,237.26,0.00),v40,z0,tPen\WObj:=wPaper;
    MoveL Offs(pOrigin,239.59,237.69,0.00),v40,z0,tPen\WObj:=wPaper;
    MoveL Offs(pOrigin,240.01,238.11,0.00),v40,z0,tPen\WObj:=wPaper;
    MoveL Offs(pOrigin,239.59,237.69,0.00),v40,z0,tPen\WObj:=wPaper;
    MoveL Offs(pOrigin,240.65,237.26,0.00),v40,z0,tPen\WObj:=wPaper;
    MoveL Offs(pOrigin,241.07,236.62,0.00),v40,z0,tPen\WObj:=wPaper;
    MoveL Offs(pOrigin,241.50,236.62,0.00),v40,z0,tPen\WObj:=wPaper;
    MoveL Offs(pOrigin,241.50,236.62,0.00),v40,z0,tPen\WObj:=wPaper;
    MoveL Offs(pOrigin,241.57,234.50,0.00),v40,z0,tPen\WObj:=wPaper;
    MoveL Offs(pOrigin,241.07,234.07,0.00),v40,z0,tPen\WObj:=wPaper;
    MoveL Offs(pOrigin,240.01,234.07,0.00),v40,z0,tPen\WObj:=wPaper;
    MoveL Offs(pOrigin,239.80,234.00,0.00),v40,z0,tPen\WObj:=wPaper;
    MoveL Offs(pOrigin,239.94,234.93,0.00),v40,z0,tPen\WObj:=wPaper;
    MoveL Offs(pOrigin,239.16,235.63,0.00),v40,z0,tPen\WObj:=wPaper;
    MoveL Offs(pOrigin,239.02,234.07,0.00),v40,z0,tPen\WObj:=wPaper;
    MoveL Offs(pOrigin,239.80,234.00,0.00),v40,fine,tPen\WObj:=wPaper;
    MoveL Offs(pOrigin,239.80,234.00,6.00),v60,z5,tPen\WObj:=wPaper;
    MoveL Offs(pOrigin,241.50,234.07,6.00),vTravel,z5,tPen\WObj:=wPaper;
    MoveL Offs(pOrigin,241.50,234.07,0.00),v60,z0,tPen\WObj:=wPaper;
    MoveL Offs(pOrigin,241.71,234.50,0.00),v40,z0,tPen\WObj:=wPaper;
    MoveL Offs(pOrigin,241.50,234.07,0.00),v40,fine,tPen\WObj:=wPaper;
    MoveL Offs(pOrigin,241.50,234.07,6.00),v60,z5,tPen\WObj:=wPaper;
    MoveL Offs(pOrigin,238.95,235.77,6.00),vTravel,z5,tPen\WObj:=wPaper;
    MoveL Offs(pOrigin,238.95,235.77,0.00),v60,z0,tPen\WObj:=wPaper;
    MoveL Offs(pOrigin,238.10,236.62,0.00),v40,fine,tPen\WObj:=wPaper;
    MoveL Offs(pOrigin,238.10,236.62,6.00),v60,z5,tPen\WObj:=wPaper;
    MoveL Offs(pOrigin,240.65,237.26,6.00),vTravel,z5,tPen\WObj:=wPaper;
    MoveL Offs(pOrigin,240.65,237.26,0.00),v60,z0,tPen\WObj:=wPaper;
    MoveL Offs(pOrigin,241.71,238.32,0.00),v40,fine,tPen\WObj:=wPaper;
    MoveL Offs(pOrigin,241.71,238.32,6.00),v60,z5,tPen\WObj:=wPaper;
    MoveL Offs(pOrigin,238.74,241.51,6.00),vTravel,z5,tPen\WObj:=wPaper;
    MoveL Offs(pOrigin,238.74,241.51,0.00),v60,z0,tPen\WObj:=wPaper;
    MoveL Offs(pOrigin,239.16,241.30,0.00),v40,z0,tPen\WObj:=wPaper;
    MoveL Offs(pOrigin,238.74,241.51,0.00),v40,fine,tPen\WObj:=wPaper;
    MoveL Offs(pOrigin,238.74,241.51,6.00),v60,z5,tPen\WObj:=wPaper;
    MoveL Offs(pOrigin,234.91,235.56,6.00),vTravel,z5,tPen\WObj:=wPaper;
    MoveL Offs(pOrigin,234.91,235.56,0.00),v60,z0,tPen\WObj:=wPaper;
    MoveL Offs(pOrigin,236.61,233.86,0.00),v40,z0,tPen\WObj:=wPaper;
    MoveL Offs(pOrigin,236.61,233.23,0.00),v40,z0,tPen\WObj:=wPaper;
    MoveL Offs(pOrigin,236.61,233.23,0.00),v40,z0,tPen\WObj:=wPaper;
    MoveL Offs(pOrigin,236.19,232.59,0.00),v40,z0,tPen\WObj:=wPaper;
    MoveL Offs(pOrigin,235.12,232.16,0.00),v40,fine,tPen\WObj:=wPaper;
    MoveL Offs(pOrigin,235.12,232.16,6.00),v60,z5,tPen\WObj:=wPaper;
    MoveL Offs(pOrigin,228.54,232.59,6.00),vTravel,z5,tPen\WObj:=wPaper;
    MoveL Offs(pOrigin,228.54,232.59,0.00),v60,z0,tPen\WObj:=wPaper;
    MoveL Offs(pOrigin,227.48,232.16,0.00),v40,z0,tPen\WObj:=wPaper;
    MoveL Offs(pOrigin,226.41,230.89,0.00),v40,z0,tPen\WObj:=wPaper;
    MoveL Offs(pOrigin,226.84,227.91,0.00),v40,z0,tPen\WObj:=wPaper;
    MoveL Offs(pOrigin,227.48,227.06,0.00),v40,fine,tPen\WObj:=wPaper;
    MoveL Offs(pOrigin,227.48,227.06,6.00),v60,z5,tPen\WObj:=wPaper;
    MoveL Offs(pOrigin,223.23,234.07,6.00),vTravel,z5,tPen\WObj:=wPaper;
    MoveL Offs(pOrigin,223.23,234.07,0.00),v60,z0,tPen\WObj:=wPaper;
    MoveL Offs(pOrigin,231.30,246.40,0.00),v40,z0,tPen\WObj:=wPaper;
    MoveL Offs(pOrigin,230.88,245.98,0.00),v40,z0,tPen\WObj:=wPaper;
    MoveL Offs(pOrigin,231.30,246.40,0.00),v40,z0,tPen\WObj:=wPaper;
    MoveL Offs(pOrigin,230.88,245.98,0.00),v40,fine,tPen\WObj:=wPaper;
    MoveL Offs(pOrigin,230.88,245.98,6.00),v60,z5,tPen\WObj:=wPaper;
    MoveL Offs(pOrigin,229.39,235.99,6.00),vTravel,z5,tPen\WObj:=wPaper;
    MoveL Offs(pOrigin,229.39,235.99,0.00),v60,z0,tPen\WObj:=wPaper;
    MoveL Offs(pOrigin,229.60,236.41,0.00),v40,z0,tPen\WObj:=wPaper;
    MoveL Offs(pOrigin,229.39,235.99,0.00),v40,fine,tPen\WObj:=wPaper;
  ENDPROC

  PROC DrawPart11()
    MoveL Offs(pOrigin,229.39,235.99,6.00),v60,z5,tPen\WObj:=wPaper;
    MoveL Offs(pOrigin,247.02,240.45,6.00),vTravel,z5,tPen\WObj:=wPaper;
    MoveL Offs(pOrigin,247.02,240.45,0.00),v60,z0,tPen\WObj:=wPaper;
    MoveL Offs(pOrigin,247.24,241.09,0.00),v40,z0,tPen\WObj:=wPaper;
    MoveL Offs(pOrigin,250.00,243.50,0.00),v40,z0,tPen\WObj:=wPaper;
    MoveL Offs(pOrigin,252.12,244.27,0.00),v40,z0,tPen\WObj:=wPaper;
    MoveL Offs(pOrigin,252.76,243.64,0.00),v40,z0,tPen\WObj:=wPaper;
    MoveL Offs(pOrigin,252.76,243.64,0.00),v40,z0,tPen\WObj:=wPaper;
    MoveL Offs(pOrigin,253.40,243.43,0.00),v40,z0,tPen\WObj:=wPaper;
    MoveL Offs(pOrigin,254.46,243.78,0.00),v40,z0,tPen\WObj:=wPaper;
    MoveL Offs(pOrigin,255.81,245.12,0.00),v40,z0,tPen\WObj:=wPaper;
    MoveL Offs(pOrigin,256.38,247.25,0.00),v40,z0,tPen\WObj:=wPaper;
    MoveL Offs(pOrigin,255.10,250.44,0.00),v40,fine,tPen\WObj:=wPaper;
    MoveL Offs(pOrigin,255.10,250.44,6.00),v60,z5,tPen\WObj:=wPaper;
    MoveL Offs(pOrigin,257.23,249.80,6.00),vTravel,z5,tPen\WObj:=wPaper;
    MoveL Offs(pOrigin,257.23,249.80,0.00),v60,z0,tPen\WObj:=wPaper;
    MoveL Offs(pOrigin,269.12,239.81,0.00),v40,fine,tPen\WObj:=wPaper;
    MoveL Offs(pOrigin,269.12,239.81,6.00),v60,z5,tPen\WObj:=wPaper;
    MoveL Offs(pOrigin,255.31,238.32,6.00),vTravel,z5,tPen\WObj:=wPaper;
    MoveL Offs(pOrigin,255.31,238.32,0.00),v60,z0,tPen\WObj:=wPaper;
    MoveL Offs(pOrigin,253.82,238.54,0.00),v40,fine,tPen\WObj:=wPaper;
    MoveL Offs(pOrigin,253.82,238.54,6.00),v60,z5,tPen\WObj:=wPaper;
    MoveL Offs(pOrigin,251.27,238.32,6.00),vTravel,z5,tPen\WObj:=wPaper;
    MoveL Offs(pOrigin,251.27,238.32,0.00),v60,z0,tPen\WObj:=wPaper;
    MoveL Offs(pOrigin,249.36,238.11,0.00),v40,z0,tPen\WObj:=wPaper;
    MoveL Offs(pOrigin,248.51,237.48,0.00),v40,fine,tPen\WObj:=wPaper;
    MoveL Offs(pOrigin,248.51,237.48,6.00),v60,z5,tPen\WObj:=wPaper;
    MoveL Offs(pOrigin,249.79,235.35,6.00),vTravel,z5,tPen\WObj:=wPaper;
    MoveL Offs(pOrigin,249.79,235.35,0.00),v60,z0,tPen\WObj:=wPaper;
    MoveL Offs(pOrigin,251.27,236.84,0.00),v40,z0,tPen\WObj:=wPaper;
    MoveL Offs(pOrigin,251.27,236.84,0.00),v40,z0,tPen\WObj:=wPaper;
    MoveL Offs(pOrigin,252.55,235.63,0.00),v40,z0,tPen\WObj:=wPaper;
    MoveL Offs(pOrigin,253.82,235.77,0.00),v40,fine,tPen\WObj:=wPaper;
    MoveL Offs(pOrigin,253.82,235.77,6.00),v60,z5,tPen\WObj:=wPaper;
    MoveL Offs(pOrigin,247.88,241.94,6.00),vTravel,z5,tPen\WObj:=wPaper;
    MoveL Offs(pOrigin,247.88,241.94,0.00),v60,z0,tPen\WObj:=wPaper;
    MoveL Offs(pOrigin,248.51,242.57,0.00),v40,z0,tPen\WObj:=wPaper;
    MoveL Offs(pOrigin,247.88,241.94,0.00),v40,fine,tPen\WObj:=wPaper;
    MoveL Offs(pOrigin,247.88,241.94,6.00),v60,z5,tPen\WObj:=wPaper;
    MoveL Offs(pOrigin,246.39,225.15,6.00),vTravel,z5,tPen\WObj:=wPaper;
    MoveL Offs(pOrigin,246.39,225.15,0.00),v60,z0,tPen\WObj:=wPaper;
    MoveL Offs(pOrigin,244.69,224.94,0.00),v40,fine,tPen\WObj:=wPaper;
    MoveL Offs(pOrigin,244.69,224.94,6.00),v60,z5,tPen\WObj:=wPaper;
    MoveL Offs(pOrigin,229.18,213.04,6.00),vTravel,z5,tPen\WObj:=wPaper;
    MoveL Offs(pOrigin,229.18,213.04,0.00),v60,z0,tPen\WObj:=wPaper;
    MoveL Offs(pOrigin,233.21,210.42,0.00),v40,z0,tPen\WObj:=wPaper;
    MoveL Offs(pOrigin,237.68,208.57,0.00),v40,z0,tPen\WObj:=wPaper;
    MoveL Offs(pOrigin,241.93,207.94,0.00),v40,z0,tPen\WObj:=wPaper;
    MoveL Offs(pOrigin,247.02,207.94,0.00),v40,z0,tPen\WObj:=wPaper;
    MoveL Offs(pOrigin,254.46,209.00,0.00),v40,z0,tPen\WObj:=wPaper;
    MoveL Offs(pOrigin,260.41,210.63,0.00),v40,z0,tPen\WObj:=wPaper;
    MoveL Offs(pOrigin,262.75,211.69,0.00),v40,z0,tPen\WObj:=wPaper;
    MoveL Offs(pOrigin,267.21,214.95,0.00),v40,fine,tPen\WObj:=wPaper;
    MoveL Offs(pOrigin,267.21,214.95,6.00),v60,z5,tPen\WObj:=wPaper;
    MoveL Offs(pOrigin,273.80,215.16,6.00),vTravel,z5,tPen\WObj:=wPaper;
    MoveL Offs(pOrigin,273.80,215.16,0.00),v60,z0,tPen\WObj:=wPaper;
    MoveL Offs(pOrigin,276.99,217.50,0.00),v40,z0,tPen\WObj:=wPaper;
    MoveL Offs(pOrigin,280.39,221.11,0.00),v40,fine,tPen\WObj:=wPaper;
    MoveL Offs(pOrigin,280.39,221.11,6.00),v60,z5,tPen\WObj:=wPaper;
    MoveL Offs(pOrigin,281.02,215.80,6.00),vTravel,z5,tPen\WObj:=wPaper;
    MoveL Offs(pOrigin,281.02,215.80,0.00),v60,z0,tPen\WObj:=wPaper;
    MoveL Offs(pOrigin,286.55,223.66,0.00),v40,z0,tPen\WObj:=wPaper;
    MoveL Offs(pOrigin,288.04,224.51,0.00),v40,z0,tPen\WObj:=wPaper;
    MoveL Offs(pOrigin,288.25,225.15,0.00),v40,z0,tPen\WObj:=wPaper;
    MoveL Offs(pOrigin,288.25,223.24,0.00),v40,z0,tPen\WObj:=wPaper;
    MoveL Offs(pOrigin,287.54,222.18,0.00),v40,z0,tPen\WObj:=wPaper;
    MoveL Offs(pOrigin,285.98,217.50,0.00),v40,z0,tPen\WObj:=wPaper;
    MoveL Offs(pOrigin,282.16,209.43,0.00),v40,z0,tPen\WObj:=wPaper;
    MoveL Offs(pOrigin,280.39,206.66,0.00),v40,z0,tPen\WObj:=wPaper;
    MoveL Offs(pOrigin,280.39,206.66,0.00),v40,z0,tPen\WObj:=wPaper;
    MoveL Offs(pOrigin,279.61,204.32,0.00),v40,z0,tPen\WObj:=wPaper;
    MoveL Offs(pOrigin,275.36,197.52,0.00),v40,z0,tPen\WObj:=wPaper;
    MoveL Offs(pOrigin,274.51,195.61,0.00),v40,z0,tPen\WObj:=wPaper;
    MoveL Offs(pOrigin,270.83,190.09,0.00),v40,z0,tPen\WObj:=wPaper;
    MoveL Offs(pOrigin,269.55,188.81,0.00),v40,z0,tPen\WObj:=wPaper;
    MoveL Offs(pOrigin,269.55,188.81,0.00),v40,z0,tPen\WObj:=wPaper;
    MoveL Offs(pOrigin,269.41,187.96,0.00),v40,z0,tPen\WObj:=wPaper;
    MoveL Offs(pOrigin,261.19,175.85,0.00),v40,z0,tPen\WObj:=wPaper;
    MoveL Offs(pOrigin,259.42,169.90,0.00),v40,z0,tPen\WObj:=wPaper;
    MoveL Offs(pOrigin,257.01,166.93,0.00),v40,z0,tPen\WObj:=wPaper;
    MoveL Offs(pOrigin,252.98,163.74,0.00),v40,fine,tPen\WObj:=wPaper;
    MoveL Offs(pOrigin,252.98,163.74,6.00),v60,z5,tPen\WObj:=wPaper;
    MoveL Offs(pOrigin,251.91,164.59,6.00),vTravel,z5,tPen\WObj:=wPaper;
    MoveL Offs(pOrigin,251.91,164.59,0.00),v60,z0,tPen\WObj:=wPaper;
    MoveL Offs(pOrigin,251.70,165.01,0.00),v40,z0,tPen\WObj:=wPaper;
    MoveL Offs(pOrigin,251.91,164.59,0.00),v40,fine,tPen\WObj:=wPaper;
    MoveL Offs(pOrigin,251.91,164.59,6.00),v60,z5,tPen\WObj:=wPaper;
    MoveL Offs(pOrigin,250.64,165.86,6.00),vTravel,z5,tPen\WObj:=wPaper;
    MoveL Offs(pOrigin,250.64,165.86,0.00),v60,z0,tPen\WObj:=wPaper;
    MoveL Offs(pOrigin,251.06,165.65,0.00),v40,z0,tPen\WObj:=wPaper;
    MoveL Offs(pOrigin,250.64,165.86,0.00),v40,fine,tPen\WObj:=wPaper;
    MoveL Offs(pOrigin,250.64,165.86,6.00),v60,z5,tPen\WObj:=wPaper;
    MoveL Offs(pOrigin,245.96,169.26,6.00),vTravel,z5,tPen\WObj:=wPaper;
    MoveL Offs(pOrigin,245.96,169.26,0.00),v60,z0,tPen\WObj:=wPaper;
    MoveL Offs(pOrigin,245.54,169.69,0.00),v40,z0,tPen\WObj:=wPaper;
    MoveL Offs(pOrigin,245.96,169.26,0.00),v40,fine,tPen\WObj:=wPaper;
    MoveL Offs(pOrigin,245.96,169.26,6.00),v60,z5,tPen\WObj:=wPaper;
    MoveL Offs(pOrigin,243.62,166.07,6.00),vTravel,z5,tPen\WObj:=wPaper;
    MoveL Offs(pOrigin,243.62,166.07,0.00),v60,z0,tPen\WObj:=wPaper;
    MoveL Offs(pOrigin,244.05,165.65,0.00),v40,z0,tPen\WObj:=wPaper;
    MoveL Offs(pOrigin,243.62,166.07,0.00),v40,z0,tPen\WObj:=wPaper;
    MoveL Offs(pOrigin,244.05,165.65,0.00),v40,z0,tPen\WObj:=wPaper;
    MoveL Offs(pOrigin,242.77,166.71,0.00),v40,z0,tPen\WObj:=wPaper;
    MoveL Offs(pOrigin,242.99,166.50,0.00),v40,z0,tPen\WObj:=wPaper;
    MoveL Offs(pOrigin,242.14,166.93,0.00),v40,z0,tPen\WObj:=wPaper;
    MoveL Offs(pOrigin,242.42,166.78,0.00),v40,z0,tPen\WObj:=wPaper;
    MoveL Offs(pOrigin,238.52,169.90,0.00),v40,z0,tPen\WObj:=wPaper;
    MoveL Offs(pOrigin,234.06,174.15,0.00),v40,z0,tPen\WObj:=wPaper;
    MoveL Offs(pOrigin,230.24,178.82,0.00),v40,z0,tPen\WObj:=wPaper;
    MoveL Offs(pOrigin,228.96,179.04,0.00),v40,fine,tPen\WObj:=wPaper;
    MoveL Offs(pOrigin,228.96,179.04,6.00),v60,z5,tPen\WObj:=wPaper;
    MoveL Offs(pOrigin,227.48,172.88,6.00),vTravel,z5,tPen\WObj:=wPaper;
    MoveL Offs(pOrigin,227.48,172.88,0.00),v60,z0,tPen\WObj:=wPaper;
    MoveL Offs(pOrigin,226.84,173.51,0.00),v40,z0,tPen\WObj:=wPaper;
    MoveL Offs(pOrigin,224.93,185.84,0.00),v40,z0,tPen\WObj:=wPaper;
    MoveL Offs(pOrigin,222.80,195.40,0.00),v40,z0,tPen\WObj:=wPaper;
    MoveL Offs(pOrigin,222.38,195.82,0.00),v40,z0,tPen\WObj:=wPaper;
    MoveL Offs(pOrigin,222.38,195.82,0.00),v40,z0,tPen\WObj:=wPaper;
    MoveL Offs(pOrigin,222.38,197.31,0.00),v40,z0,tPen\WObj:=wPaper;
    MoveL Offs(pOrigin,220.68,205.39,0.00),v40,z0,tPen\WObj:=wPaper;
  ENDPROC

